    movel([0.342925, -1.240601, -2.657500, -0.814287, 1.570796, 1.913721],accel_mss,speed_ms,0,blend_radius_m)
    movel([0.344869, -1.239133, -2.658265, -0.814990, 1.570796, 1.915665],accel_mss,speed_ms,0,blend_radius_m)
    movel([0.348721, -1.236542, -2.659609, -0.816237, 1.570796, 1.919517],accel_mss,speed_ms,0,blend_radius_m)
    movel([0.352271, -1.234571, -2.660626, -0.817191, 1.570796, 1.923067],accel_mss,speed_ms,0,blend_radius_m)
    movel([0.353507, -1.234027, -2.660906, -0.817455, 1.570796, 1.924303],accel_mss,speed_ms,0,blend_radius_m)
    movel([0.354725, -1.233660, -2.661095, -0.817634, 1.570796, 1.925522],accel_mss,speed_ms,0,blend_radius_m)
    movel([0.355376, -1.233628, -2.661112, -0.817650, 1.570796, 1.926173],accel_mss,speed_ms,0,blend_radius_m)
    movel([0.355877, -1.233849, -2.660998, -0.817542, 1.570796, 1.926673],accel_mss,speed_ms,0,blend_radius_m)
    movel([0.356080, -1.234279, -2.660777, -0.817333, 1.570796, 1.926876],accel_mss,speed_ms,0,blend_radius_m)
    movel([0.355956, -1.234871, -2.660472, -0.817046, 1.570796, 1.926752],accel_mss,speed_ms,0,blend_radius_m)
    movel([0.355650, -1.235547, -2.660124, -0.816719, 1.570796, 1.926446],accel_mss,speed_ms,0,blend_radius_m)
    movel([0.353652, -1.236176, -2.659798, -0.816414, 1.570796, 1.924449],accel_mss,speed_ms,0,blend_radius_m)
    movel([0.351697, -1.236940, -2.659404, -0.816046, 1.570796, 1.922493],accel_mss,speed_ms,0,blend_radius_m)
    movel([0.349633, -1.238027, -2.658840, -0.815522, 1.570796, 1.920429],accel_mss,speed_ms,0,blend_radius_m)
    movel([0.347319, -1.239519, -2.658064, -0.814805, 1.570796, 1.918116],accel_mss,speed_ms,0,blend_radius_m)
    movel([0.344599, -1.241515, -2.657023, -0.813851, 1.570796, 1.915395],accel_mss,speed_ms,0,blend_radius_m)
    movel([0.342464, -1.243303, -2.656086, -0.813000, 1.570796, 1.913260],accel_mss,speed_ms,0,blend_radius_m)
    movel([0.341814, -1.243974, -2.655733, -0.812682, 1.570796, 1.912611],accel_mss,speed_ms,0,blend_radius_m)
    movel([0.341272, -1.244705, -2.655349, -0.812336, 1.570796, 1.912068],accel_mss,speed_ms,0,blend_radius_m)
    movel([0.340309, -1.246556, -2.654371, -0.811462, 1.570796, 1.911105],accel_mss,speed_ms,0,blend_radius_m)
    movel([0.337343, -1.254210, -2.650287, -0.807892, 1.570796, 1.908139],accel_mss,speed_ms,0,blend_radius_m)
    movel([0.336811, -1.255318, -2.649690, -0.807381, 1.570796, 1.907607],accel_mss,speed_ms,0,blend_radius_m)
    movel([0.334705, -1.258850, -2.647777, -0.805762, 1.570796, 1.905501],accel_mss,speed_ms,0,blend_radius_m)
    movel([0.333378, -1.260708, -2.646764, -0.804917, 1.570796, 1.904174],accel_mss,speed_ms,0,blend_radius_m)
    movel([0.331727, -1.262673, -2.645689, -0.804027, 1.570796, 1.902523],accel_mss,speed_ms,0,blend_radius_m)
    movel([0.329183, -1.265435, -2.644170, -0.802785, 1.570796, 1.899980],accel_mss,speed_ms,0,blend_radius_m)
    movel([0.328186, -1.266665, -2.643490, -0.802234, 1.570796, 1.898982],accel_mss,speed_ms,0,blend_radius_m)
    movel([0.327796, -1.267344, -2.643114, -0.801931, 1.570796, 1.898592],accel_mss,speed_ms,0,blend_radius_m)
    movel([0.324763, -1.273372, -2.639750, -0.799266, 1.570796, 1.895559],accel_mss,speed_ms,0,blend_radius_m)
    movel([0.324383, -1.274130, -2.639324, -0.798934, 1.570796, 1.895179],accel_mss,speed_ms,0,blend_radius_m)
    movel([0.324022, -1.275035, -2.638815, -0.798539, 1.570796, 1.894818],accel_mss,speed_ms,0,blend_radius_m)
    movel([0.323870, -1.275151, -2.638750, -0.798489, 1.570796, 1.894666],accel_mss,speed_ms,0,blend_radius_m)
    movel([0.320813, -1.276074, -2.638228, -0.798087, 1.570796, 1.891609],accel_mss,speed_ms,0,blend_radius_m)
    movel([0.319322, -1.276354, -2.638070, -0.797965, 1.570796, 1.890119],accel_mss,speed_ms,0,blend_radius_m)
    movel([0.317735, -1.276515, -2.637979, -0.797895, 1.570796, 1.888532],accel_mss,speed_ms,0,blend_radius_m)
    movel([0.316753, -1.276438, -2.638023, -0.797928, 1.570796, 1.887549],accel_mss,speed_ms,0,blend_radius_m)
    movel([0.316033, -1.276098, -2.638215, -0.798076, 1.570796, 1.886829],accel_mss,speed_ms,0,blend_radius_m)
    movel([0.315335, -1.275398, -2.638610, -0.798381, 1.570796, 1.886132],accel_mss,speed_ms,0,blend_radius_m)
    movel([0.314818, -1.274603, -2.639058, -0.798728, 1.570796, 1.885614],accel_mss,speed_ms,0,blend_radius_m)
    movel([0.314451, -1.273698, -2.639567, -0.799124, 1.570796, 1.885248],accel_mss,speed_ms,0,blend_radius_m)
    movel([0.314212, -1.272638, -2.640162, -0.799588, 1.570796, 1.885009],accel_mss,speed_ms,0,blend_radius_m)
    movel([0.314114, -1.271502, -2.640799, -0.800088, 1.570796, 1.884911],accel_mss,speed_ms,0,blend_radius_m)
    movel([0.314331, -1.268769, -2.642323, -0.801297, 1.570796, 1.885128],accel_mss,speed_ms,0,blend_radius_m)
    movel([0.315111, -1.265451, -2.644161, -0.802778, 1.570796, 1.885907],accel_mss,speed_ms,0,blend_radius_m)
    movel([0.315866, -1.263112, -2.645448, -0.803829, 1.570796, 1.886662],accel_mss,speed_ms,0,blend_radius_m)
    movel([0.316606, -1.261364, -2.646406, -0.804619, 1.570796, 1.887402],accel_mss,speed_ms,0,blend_radius_m)
    movel([0.317785, -1.259161, -2.647608, -0.805620, 1.570796, 1.888582],accel_mss,speed_ms,0,blend_radius_m)
    movel([0.320612, -1.254305, -2.650236, -0.807848, 1.570796, 1.891408],accel_mss,speed_ms,0,blend_radius_m)
    movel([0.326605, -1.243916, -2.655764, -0.812709, 1.570796, 1.897401],accel_mss,speed_ms,0,blend_radius_m)
    movel([0.327796, -1.241515, -2.657023, -0.813851, 1.570796, 1.898593],accel_mss,speed_ms,0,blend_radius_m)
    movel([0.328653, -1.239347, -2.658154, -0.814888, 1.570796, 1.899449],accel_mss,speed_ms,0,blend_radius_m)
    movel([0.329234, -1.237182, -2.659278, -0.815929, 1.570796, 1.900030],accel_mss,speed_ms,0,blend_radius_m)
    movel([0.329337, -1.235501, -2.660147, -0.816741, 1.570796, 1.900134],accel_mss,speed_ms,0,blend_radius_m)
    movel([0.328959, -1.233999, -2.660921, -0.817469, 1.570796, 1.899755],accel_mss,speed_ms,0,blend_radius_m)
    movel([0.327249, -1.231057, -2.662428, -0.818903, 1.570796, 1.898045],accel_mss,speed_ms,0,blend_radius_m)
    movel([0.327023, -1.230500, -2.662713, -0.819176, 1.570796, 1.897820],accel_mss,speed_ms,0,blend_radius_m)
    movel([0.327053, -1.229355, -2.663296, -0.819738, 1.570796, 1.897849],accel_mss,speed_ms,0,blend_radius_m)
    movel([0.327307, -1.228564, -2.663698, -0.820126, 1.570796, 1.898103],accel_mss,speed_ms,0,blend_radius_m)
    movel([0.328348, -1.226520, -2.664734, -0.821135, 1.570796, 1.899144],accel_mss,speed_ms,0,blend_radius_m)
    movel([0.330098, -1.223921, -2.666045, -0.822424, 1.570796, 1.900894],accel_mss,speed_ms,0,blend_radius_m)
    movel([0.332667, -1.220640, -2.667687, -0.824062, 1.570796, 1.903464],accel_mss,speed_ms,0,blend_radius_m)
    movel([0.335094, -1.217632, -2.669182, -0.825575, 1.570796, 1.905891],accel_mss,speed_ms,0,blend_radius_m)
    movel([0.338739, -1.212850, -2.671539, -0.828001, 1.570796, 1.909536],accel_mss,speed_ms,0,blend_radius_m)
    movel([0.338922, -1.212365, -2.671776, -0.828248, 1.570796, 1.909718],accel_mss,speed_ms,0,blend_radius_m)
    movel([0.338575, -1.212129, -2.671891, -0.828368, 1.570796, 1.909372],accel_mss,speed_ms,0,blend_radius_m)
    movel([0.338364, -1.212140, -2.671886, -0.828363, 1.570796, 1.909160],accel_mss,speed_ms,0,blend_radius_m)
    movel([0.337571, -1.212519, -2.671701, -0.828169, 1.570796, 1.908368],accel_mss,speed_ms,0,blend_radius_m)
    movel([0.335837, -1.213970, -2.670989, -0.827430, 1.570796, 1.906634],accel_mss,speed_ms,0,blend_radius_m)
    movel([0.334072, -1.215612, -2.670181, -0.826596, 1.570796, 1.904868],accel_mss,speed_ms,0,blend_radius_m)
    movel([0.332776, -1.217039, -2.669476, -0.825874, 1.570796, 1.903572],accel_mss,speed_ms,0,blend_radius_m)
    movel([0.331388, -1.218851, -2.668578, -0.824960, 1.570796, 1.902184],accel_mss,speed_ms,0,blend_radius_m)
    movel([0.328906, -1.222329, -2.666843, -0.823217, 1.570796, 1.899703],accel_mss,speed_ms,0,blend_radius_m)
    movel([0.325279, -1.227661, -2.664156, -0.820571, 1.570796, 1.896075],accel_mss,speed_ms,0,blend_radius_m)
    movel([0.324263, -1.229633, -2.663155, -0.819601, 1.570796, 1.895059],accel_mss,speed_ms,0,blend_radius_m)
    movel([0.323797, -1.231289, -2.662310, -0.818790, 1.570796, 1.894593],accel_mss,speed_ms,0,blend_radius_m)
    movel([0.323833, -1.232893, -2.661489, -0.818007, 1.570796, 1.894629],accel_mss,speed_ms,0,blend_radius_m)
    movel([0.324369, -1.234718, -2.660551, -0.817120, 1.570796, 1.895165],accel_mss,speed_ms,0,blend_radius_m)
    movel([0.324847, -1.236239, -2.659766, -0.816384, 1.570796, 1.895643],accel_mss,speed_ms,0,blend_radius_m)
    movel([0.325003, -1.237579, -2.659073, -0.815738, 1.570796, 1.895799],accel_mss,speed_ms,0,blend_radius_m)
    movel([0.324852, -1.238985, -2.658342, -0.815062, 1.570796, 1.895648],accel_mss,speed_ms,0,blend_radius_m)
    movel([0.324386, -1.240693, -2.657452, -0.814244, 1.570796, 1.895183],accel_mss,speed_ms,0,blend_radius_m)
    movel([0.322806, -1.244813, -2.655291, -0.812284, 1.570796, 1.893602],accel_mss,speed_ms,0,blend_radius_m)
    movel([0.320559, -1.249674, -2.652716, -0.809999, 1.570796, 1.891355],accel_mss,speed_ms,0,blend_radius_m)
    movel([0.317904, -1.254769, -2.649986, -0.807634, 1.570796, 1.888700],accel_mss,speed_ms,0,blend_radius_m)
    movel([0.313546, -1.262291, -2.645898, -0.804199, 1.570796, 1.884343],accel_mss,speed_ms,0,blend_radius_m)
    movel([0.312665, -1.264271, -2.644811, -0.803307, 1.570796, 1.883462],accel_mss,speed_ms,0,blend_radius_m)
    movel([0.312161, -1.266203, -2.643745, -0.802441, 1.570796, 1.882958],accel_mss,speed_ms,0,blend_radius_m)
    movel([0.311861, -1.268682, -2.642371, -0.801336, 1.570796, 1.882658],accel_mss,speed_ms,0,blend_radius_m)
    movel([0.311715, -1.271688, -2.640695, -0.800006, 1.570796, 1.882512],accel_mss,speed_ms,0,blend_radius_m)
    movel([0.311845, -1.273631, -2.639605, -0.799153, 1.570796, 1.882642],accel_mss,speed_ms,0,blend_radius_m)
    movel([0.312275, -1.275014, -2.638826, -0.798548, 1.570796, 1.883071],accel_mss,speed_ms,0,blend_radius_m)
    movel([0.313063, -1.276155, -2.638183, -0.798051, 1.570796, 1.883860],accel_mss,speed_ms,0,blend_radius_m)
    movel([0.313700, -1.276690, -2.637880, -0.797819, 1.570796, 1.884496],accel_mss,speed_ms,0,blend_radius_m)
    movel([0.314469, -1.277118, -2.637638, -0.797633, 1.570796, 1.885265],accel_mss,speed_ms,0,blend_radius_m)
    movel([0.316829, -1.277817, -2.637241, -0.797330, 1.570796, 1.887625],accel_mss,speed_ms,0,blend_radius_m)
    movel([0.318196, -1.277977, -2.637151, -0.797261, 1.570796, 1.888993],accel_mss,speed_ms,0,blend_radius_m)
    movel([0.319769, -1.277907, -2.637190, -0.797291, 1.570796, 1.890565],accel_mss,speed_ms,0,blend_radius_m)
    movel([0.321417, -1.277620, -2.637353, -0.797415, 1.570796, 1.892213],accel_mss,speed_ms,0,blend_radius_m)
    movel([0.323020, -1.277130, -2.637631, -0.797628, 1.570796, 1.893817],accel_mss,speed_ms,0,blend_radius_m)
    movel([0.324631, -1.276538, -2.637966, -0.797885, 1.570796, 1.895428],accel_mss,speed_ms,0,blend_radius_m)
    movel([0.325024, -1.276490, -2.637993, -0.797906, 1.570796, 1.895820],accel_mss,speed_ms,0,blend_radius_m)
    movel([0.325205, -1.276670, -2.637892, -0.797828, 1.570796, 1.896001],accel_mss,speed_ms,0,blend_radius_m)
    movel([0.325256, -1.277465, -2.637442, -0.797483, 1.570796, 1.896052],accel_mss,speed_ms,0,blend_radius_m)
    movel([0.325263, -1.278170, -2.637041, -0.797178, 1.570796, 1.896059],accel_mss,speed_ms,0,blend_radius_m)
    movel([0.325097, -1.278682, -2.636751, -0.796957, 1.570796, 1.895893],accel_mss,speed_ms,0,blend_radius_m)
    movel([0.324858, -1.278895, -2.636630, -0.796865, 1.570796, 1.895654],accel_mss,speed_ms,0,blend_radius_m)
    movel([0.323615, -1.279507, -2.636281, -0.796601, 1.570796, 1.894411],accel_mss,speed_ms,0,blend_radius_m)
    movel([0.322799, -1.279816, -2.636106, -0.796468, 1.570796, 1.893596],accel_mss,speed_ms,0,blend_radius_m)
    movel([0.322396, -1.281444, -2.635176, -0.795769, 1.570796, 1.893192],accel_mss,speed_ms,0,blend_radius_m)
    movel([0.321882, -1.283464, -2.634019, -0.794906, 1.570796, 1.892679],accel_mss,speed_ms,0,blend_radius_m)
    movel([0.321665, -1.283948, -2.633741, -0.794700, 1.570796, 1.892462],accel_mss,speed_ms,0,blend_radius_m)
    movel([0.321328, -1.284205, -2.633593, -0.794591, 1.570796, 1.892124],accel_mss,speed_ms,0,blend_radius_m)
    movel([0.320496, -1.284406, -2.633477, -0.794506, 1.570796, 1.891293],accel_mss,speed_ms,0,blend_radius_m)
    movel([0.319352, -1.284617, -2.633356, -0.794416, 1.570796, 1.890149],accel_mss,speed_ms,0,blend_radius_m)
    movel([0.319034, -1.286067, -2.632519, -0.793802, 1.570796, 1.889831],accel_mss,speed_ms,0,blend_radius_m)
    movel([0.318968, -1.286670, -2.632171, -0.793548, 1.570796, 1.889764],accel_mss,speed_ms,0,blend_radius_m)
    movel([0.318918, -1.289142, -2.630737, -0.792510, 1.570796, 1.889714],accel_mss,speed_ms,0,blend_radius_m)
    movel([0.317168, -1.289744, -2.630387, -0.792258, 1.570796, 1.887964],accel_mss,speed_ms,0,blend_radius_m)
    movel([0.316818, -1.289909, -2.630291, -0.792189, 1.570796, 1.887614],accel_mss,speed_ms,0,blend_radius_m)
    movel([0.316442, -1.290304, -2.630061, -0.792024, 1.570796, 1.887238],accel_mss,speed_ms,0,blend_radius_m)
    movel([0.316388, -1.290467, -2.629966, -0.791956, 1.570796, 1.887184],accel_mss,speed_ms,0,blend_radius_m)
    movel([0.316505, -1.290778, -2.629785, -0.791827, 1.570796, 1.887301],accel_mss,speed_ms,0,blend_radius_m)
    movel([0.317002, -1.290765, -2.629792, -0.791832, 1.570796, 1.887798],accel_mss,speed_ms,0,blend_radius_m)
    movel([0.319686, -1.289953, -2.630265, -0.792171, 1.570796, 1.890482],accel_mss,speed_ms,0,blend_radius_m)
    movel([0.320071, -1.289692, -2.630418, -0.792280, 1.570796, 1.890868],accel_mss,speed_ms,0,blend_radius_m)
    movel([0.320223, -1.289323, -2.630632, -0.792434, 1.570796, 1.891019],accel_mss,speed_ms,0,blend_radius_m)
    movel([0.320249, -1.289064, -2.630782, -0.792542, 1.570796, 1.891046],accel_mss,speed_ms,0,blend_radius_m)
    movel([0.320099, -1.286560, -2.632235, -0.793594, 1.570796, 1.890895],accel_mss,speed_ms,0,blend_radius_m)
    movel([0.320118, -1.286092, -2.632505, -0.793792, 1.570796, 1.890915],accel_mss,speed_ms,0,blend_radius_m)
    movel([0.320281, -1.285655, -2.632757, -0.793977, 1.570796, 1.891077],accel_mss,speed_ms,0,blend_radius_m)
    movel([0.320489, -1.285544, -2.632822, -0.794024, 1.570796, 1.891285],accel_mss,speed_ms,0,blend_radius_m)
    movel([0.321725, -1.285126, -2.633063, -0.794201, 1.570796, 1.892522],accel_mss,speed_ms,0,blend_radius_m)
    movel([0.322077, -1.284938, -2.633171, -0.794280, 1.570796, 1.892874],accel_mss,speed_ms,0,blend_radius_m)
    movel([0.322644, -1.284448, -2.633453, -0.794488, 1.570796, 1.893440],accel_mss,speed_ms,0,blend_radius_m)
    movel([0.322831, -1.284146, -2.633627, -0.794616, 1.570796, 1.893627],accel_mss,speed_ms,0,blend_radius_m)
    movel([0.323519, -1.281183, -2.635325, -0.795880, 1.570796, 1.894315],accel_mss,speed_ms,0,blend_radius_m)
    movel([0.323687, -1.280709, -2.635596, -0.796084, 1.570796, 1.894484],accel_mss,speed_ms,0,blend_radius_m)
    movel([0.323943, -1.280423, -2.635759, -0.796206, 1.570796, 1.894740],accel_mss,speed_ms,0,blend_radius_m)
    movel([0.324430, -1.280152, -2.635914, -0.796323, 1.570796, 1.895227],accel_mss,speed_ms,0,blend_radius_m)
    movel([0.325816, -1.279294, -2.636403, -0.796693, 1.570796, 1.896612],accel_mss,speed_ms,0,blend_radius_m)
    movel([0.326505, -1.278741, -2.636717, -0.796931, 1.570796, 1.897301],accel_mss,speed_ms,0,blend_radius_m)
    movel([0.326437, -1.275734, -2.638420, -0.798234, 1.570796, 1.897233],accel_mss,speed_ms,0,blend_radius_m)
    movel([0.327765, -1.274947, -2.638865, -0.798578, 1.570796, 1.898561],accel_mss,speed_ms,0,blend_radius_m)
    movel([0.328461, -1.274549, -2.639089, -0.798751, 1.570796, 1.899257],accel_mss,speed_ms,0,blend_radius_m)
    movel([0.335186, -1.270304, -2.641468, -0.800617, 1.570796, 1.905982],accel_mss,speed_ms,0,blend_radius_m)
    movel([0.334839, -1.272294, -2.640355, -0.799740, 1.570796, 1.905635],accel_mss,speed_ms,0,blend_radius_m)
    movel([0.332590, -1.273380, -2.639746, -0.799263, 1.570796, 1.903387],accel_mss,speed_ms,0,blend_radius_m)
    movel([0.330282, -1.274619, -2.639049, -0.798721, 1.570796, 1.901079],accel_mss,speed_ms,0,blend_radius_m)
    movel([0.330077, -1.274797, -2.638949, -0.798643, 1.570796, 1.900873],accel_mss,speed_ms,0,blend_radius_m)
    movel([0.329178, -1.276573, -2.637946, -0.797870, 1.570796, 1.899974],accel_mss,speed_ms,0,blend_radius_m)
    movel([0.328530, -1.277951, -2.637165, -0.797272, 1.570796, 1.899326],accel_mss,speed_ms,0,blend_radius_m)
    movel([0.328008, -1.278732, -2.636722, -0.796935, 1.570796, 1.898804],accel_mss,speed_ms,0,blend_radius_m)
    movel([0.327346, -1.279338, -2.636377, -0.796673, 1.570796, 1.898142],accel_mss,speed_ms,0,blend_radius_m)
    movel([0.326248, -1.280043, -2.635976, -0.796370, 1.570796, 1.897044],accel_mss,speed_ms,0,blend_radius_m)
    movel([0.324771, -1.280902, -2.635486, -0.796001, 1.570796, 1.895567],accel_mss,speed_ms,0,blend_radius_m)
    movel([0.323793, -1.283902, -2.633767, -0.794720, 1.570796, 1.894589],accel_mss,speed_ms,0,blend_radius_m)
    movel([0.323562, -1.284445, -2.633455, -0.794489, 1.570796, 1.894359],accel_mss,speed_ms,0,blend_radius_m)
    movel([0.322925, -1.285601, -2.632788, -0.793999, 1.570796, 1.893721],accel_mss,speed_ms,0,blend_radius_m)
    movel([0.322536, -1.286003, -2.632556, -0.793830, 1.570796, 1.893333],accel_mss,speed_ms,0,blend_radius_m)
    movel([0.320605, -1.287668, -2.631593, -0.793128, 1.570796, 1.891402],accel_mss,speed_ms,0,blend_radius_m)
    movel([0.320516, -1.287805, -2.631514, -0.793070, 1.570796, 1.891312],accel_mss,speed_ms,0,blend_radius_m)
    movel([0.320529, -1.288423, -2.631155, -0.792811, 1.570796, 1.891325],accel_mss,speed_ms,0,blend_radius_m)
    movel([0.320576, -1.288693, -2.630998, -0.792698, 1.570796, 1.891372],accel_mss,speed_ms,0,blend_radius_m)
    movel([0.320625, -1.291004, -2.629653, -0.791733, 1.570796, 1.891421],accel_mss,speed_ms,0,blend_radius_m)
    movel([0.320771, -1.291367, -2.629441, -0.791582, 1.570796, 1.891568],accel_mss,speed_ms,0,blend_radius_m)
    movel([0.321046, -1.291426, -2.629406, -0.791557, 1.570796, 1.891842],accel_mss,speed_ms,0,blend_radius_m)
    movel([0.321425, -1.291226, -2.629523, -0.791640, 1.570796, 1.892222],accel_mss,speed_ms,0,blend_radius_m)
    movel([0.322031, -1.290877, -2.629727, -0.791785, 1.570796, 1.892827],accel_mss,speed_ms,0,blend_radius_m)
    movel([0.317945, -1.294449, -2.627633, -0.790307, 1.570796, 1.888741],accel_mss,speed_ms,0,blend_radius_m)
    movel([0.314705, -1.297568, -2.625792, -0.789029, 1.570796, 1.885501],accel_mss,speed_ms,0,blend_radius_m)
    movel([0.311613, -1.300747, -2.623903, -0.787739, 1.570796, 1.882409],accel_mss,speed_ms,0,blend_radius_m)
    movel([0.309536, -1.303153, -2.622464, -0.786772, 1.570796, 1.880332],accel_mss,speed_ms,0,blend_radius_m)
    movel([0.307881, -1.305516, -2.621043, -0.785829, 1.570796, 1.878677],accel_mss,speed_ms,0,blend_radius_m)
    movel([0.307303, -1.306574, -2.620406, -0.785410, 1.570796, 1.878099],accel_mss,speed_ms,0,blend_radius_m)
    movel([0.306855, -1.307631, -2.619766, -0.784992, 1.570796, 1.877651],accel_mss,speed_ms,0,blend_radius_m)
    movel([0.306618, -1.308486, -2.619248, -0.784655, 1.570796, 1.877415],accel_mss,speed_ms,0,blend_radius_m)
    movel([0.306533, -1.309299, -2.618754, -0.784335, 1.570796, 1.877329],accel_mss,speed_ms,0,blend_radius_m)
    movel([0.306634, -1.309898, -2.618390, -0.784100, 1.570796, 1.877431],accel_mss,speed_ms,0,blend_radius_m)
    movel([0.306944, -1.310362, -2.618108, -0.783919, 1.570796, 1.877741],accel_mss,speed_ms,0,blend_radius_m)
    movel([0.307420, -1.310668, -2.617922, -0.783799, 1.570796, 1.878216],accel_mss,speed_ms,0,blend_radius_m)
    movel([0.307844, -1.310614, -2.617955, -0.783820, 1.570796, 1.878640],accel_mss,speed_ms,0,blend_radius_m)
    movel([0.308283, -1.310234, -2.618186, -0.783969, 1.570796, 1.879079],accel_mss,speed_ms,0,blend_radius_m)
    movel([0.309618, -1.308138, -2.619459, -0.784792, 1.570796, 1.880414],accel_mss,speed_ms,0,blend_radius_m)
    movel([0.309710, -1.308359, -2.619325, -0.784705, 1.570796, 1.880506],accel_mss,speed_ms,0,blend_radius_m)
    movel([0.309632, -1.308862, -2.619020, -0.784507, 1.570796, 1.880428],accel_mss,speed_ms,0,blend_radius_m)
    movel([0.309835, -1.310236, -2.618185, -0.783968, 1.570796, 1.880632],accel_mss,speed_ms,0,blend_radius_m)
    movel([0.310053, -1.310680, -2.617915, -0.783795, 1.570796, 1.880849],accel_mss,speed_ms,0,blend_radius_m)
    movel([0.310331, -1.310909, -2.617775, -0.783705, 1.570796, 1.881127],accel_mss,speed_ms,0,blend_radius_m)
    movel([0.310697, -1.310970, -2.617737, -0.783681, 1.570796, 1.881493],accel_mss,speed_ms,0,blend_radius_m)
    movel([0.311102, -1.310852, -2.617810, -0.783727, 1.570796, 1.881898],accel_mss,speed_ms,0,blend_radius_m)
    movel([0.311497, -1.310578, -2.617977, -0.783834, 1.570796, 1.882293],accel_mss,speed_ms,0,blend_radius_m)
    movel([0.313004, -1.308779, -2.619070, -0.784539, 1.570796, 1.883800],accel_mss,speed_ms,0,blend_radius_m)
    movel([0.314562, -1.306982, -2.620159, -0.785248, 1.570796, 1.885358],accel_mss,speed_ms,0,blend_radius_m)
    movel([0.316271, -1.305388, -2.621121, -0.785880, 1.570796, 1.887067],accel_mss,speed_ms,0,blend_radius_m)
    movel([0.318253, -1.303895, -2.622019, -0.786475, 1.570796, 1.889049],accel_mss,speed_ms,0,blend_radius_m)
    movel([0.320643, -1.302395, -2.622918, -0.787076, 1.570796, 1.891440],accel_mss,speed_ms,0,blend_radius_m)
    movel([0.322090, -1.301513, -2.623446, -0.787431, 1.570796, 1.892887],accel_mss,speed_ms,0,blend_radius_m)
    movel([0.323181, -1.300731, -2.623912, -0.787746, 1.570796, 1.893977],accel_mss,speed_ms,0,blend_radius_m)
    movel([0.324024, -1.299978, -2.624361, -0.788050, 1.570796, 1.894820],accel_mss,speed_ms,0,blend_radius_m)
    movel([0.324700, -1.299185, -2.624833, -0.788371, 1.570796, 1.895496],accel_mss,speed_ms,0,blend_radius_m)
    movel([0.325241, -1.298267, -2.625378, -0.788744, 1.570796, 1.896038],accel_mss,speed_ms,0,blend_radius_m)
    movel([0.326301, -1.295864, -2.626800, -0.789725, 1.570796, 1.897097],accel_mss,speed_ms,0,blend_radius_m)
    movel([0.327337, -1.293401, -2.628249, -0.790739, 1.570796, 1.898134],accel_mss,speed_ms,0,blend_radius_m)
    movel([0.327468, -1.292744, -2.628635, -0.791011, 1.570796, 1.898264],accel_mss,speed_ms,0,blend_radius_m)
    movel([0.327010, -1.292596, -2.628721, -0.791072, 1.570796, 1.897806],accel_mss,speed_ms,0,blend_radius_m)
    movel([0.326728, -1.292738, -2.628638, -0.791013, 1.570796, 1.897524],accel_mss,speed_ms,0,blend_radius_m)
    movel([0.326507, -1.292983, -2.628494, -0.790911, 1.570796, 1.897303],accel_mss,speed_ms,0,blend_radius_m)
    movel([0.326260, -1.293466, -2.628211, -0.790712, 1.570796, 1.897057],accel_mss,speed_ms,0,blend_radius_m)
    movel([0.324268, -1.298014, -2.625528, -0.788847, 1.570796, 1.895064],accel_mss,speed_ms,0,blend_radius_m)
    movel([0.323726, -1.298957, -2.624968, -0.788464, 1.570796, 1.894522],accel_mss,speed_ms,0,blend_radius_m)
    movel([0.323219, -1.299594, -2.624590, -0.788205, 1.570796, 1.894016],accel_mss,speed_ms,0,blend_radius_m)
    movel([0.322852, -1.299911, -2.624401, -0.788077, 1.570796, 1.893648],accel_mss,speed_ms,0,blend_radius_m)
    movel([0.320257, -1.301603, -2.623392, -0.787394, 1.570796, 1.891053],accel_mss,speed_ms,0,blend_radius_m)
    movel([0.317454, -1.303416, -2.622306, -0.786667, 1.570796, 1.888250],accel_mss,speed_ms,0,blend_radius_m)
    movel([0.315089, -1.305277, -2.621188, -0.785924, 1.570796, 1.885885],accel_mss,speed_ms,0,blend_radius_m)
    movel([0.313132, -1.307206, -2.620023, -0.785159, 1.570796, 1.883929],accel_mss,speed_ms,0,blend_radius_m)
    movel([0.311547, -1.309229, -2.618797, -0.784363, 1.570796, 1.882344],accel_mss,speed_ms,0,blend_radius_m)
    movel([0.311164, -1.309800, -2.618450, -0.784139, 1.570796, 1.881960],accel_mss,speed_ms,0,blend_radius_m)
    movel([0.310958, -1.309434, -2.618672, -0.784282, 1.570796, 1.881754],accel_mss,speed_ms,0,blend_radius_m)
    movel([0.310806, -1.308882, -2.619008, -0.784499, 1.570796, 1.881602],accel_mss,speed_ms,0,blend_radius_m)
    movel([0.310862, -1.308093, -2.619487, -0.784810, 1.570796, 1.881658],accel_mss,speed_ms,0,blend_radius_m)
    movel([0.311103, -1.307181, -2.620039, -0.785170, 1.570796, 1.881900],accel_mss,speed_ms,0,blend_radius_m)
    movel([0.311870, -1.305620, -2.620981, -0.785788, 1.570796, 1.882666],accel_mss,speed_ms,0,blend_radius_m)
    movel([0.312202, -1.305169, -2.621253, -0.785967, 1.570796, 1.882998],accel_mss,speed_ms,0,blend_radius_m)
    movel([0.313355, -1.304117, -2.621885, -0.786386, 1.570796, 1.884152],accel_mss,speed_ms,0,blend_radius_m)
    movel([0.314742, -1.303078, -2.622509, -0.786802, 1.570796, 1.885538],accel_mss,speed_ms,0,blend_radius_m)
    movel([0.316222, -1.302150, -2.623065, -0.787174, 1.570796, 1.887019],accel_mss,speed_ms,0,blend_radius_m)
    movel([0.317816, -1.301322, -2.623560, -0.787507, 1.570796, 1.888613],accel_mss,speed_ms,0,blend_radius_m)
    movel([0.321143, -1.299907, -2.624404, -0.788079, 1.570796, 1.891939],accel_mss,speed_ms,0,blend_radius_m)
    movel([0.321780, -1.299609, -2.624581, -0.788199, 1.570796, 1.892576],accel_mss,speed_ms,0,blend_radius_m)
    movel([0.322460, -1.299066, -2.624903, -0.788419, 1.570796, 1.893257],accel_mss,speed_ms,0,blend_radius_m)
    movel([0.322781, -1.298643, -2.625155, -0.788591, 1.570796, 1.893577],accel_mss,speed_ms,0,blend_radius_m)
    movel([0.325964, -1.293186, -2.628375, -0.790828, 1.570796, 1.896760],accel_mss,speed_ms,0,blend_radius_m)
    movel([0.326690, -1.291543, -2.629337, -0.791508, 1.570796, 1.897486],accel_mss,speed_ms,0,blend_radius_m)
    movel([0.326759, -1.291157, -2.629563, -0.791669, 1.570796, 1.897555],accel_mss,speed_ms,0,blend_radius_m)
    movel([0.326656, -1.290909, -2.629708, -0.791772, 1.570796, 1.897453],accel_mss,speed_ms,0,blend_radius_m)
    movel([0.326423, -1.290864, -2.629734, -0.791791, 1.570796, 1.897220],accel_mss,speed_ms,0,blend_radius_m)
    movel([0.326121, -1.291020, -2.629643, -0.791726, 1.570796, 1.896918],accel_mss,speed_ms,0,blend_radius_m)
    movel([0.325974, -1.291191, -2.629543, -0.791655, 1.570796, 1.896770],accel_mss,speed_ms,0,blend_radius_m)
    movel([0.325499, -1.292006, -2.629067, -0.791316, 1.570796, 1.896296],accel_mss,speed_ms,0,blend_radius_m)
    movel([0.322492, -1.297479, -2.625845, -0.789065, 1.570796, 1.893288],accel_mss,speed_ms,0,blend_radius_m)
    movel([0.321971, -1.298129, -2.625460, -0.788800, 1.570796, 1.892767],accel_mss,speed_ms,0,blend_radius_m)
    movel([0.321361, -1.298657, -2.625147, -0.788586, 1.570796, 1.892157],accel_mss,speed_ms,0,blend_radius_m)
    movel([0.320584, -1.299114, -2.624875, -0.788400, 1.570796, 1.891380],accel_mss,speed_ms,0,blend_radius_m)
    movel([0.319549, -1.299559, -2.624610, -0.788219, 1.570796, 1.890346],accel_mss,speed_ms,0,blend_radius_m)
    movel([0.317931, -1.300249, -2.624200, -0.787940, 1.570796, 1.888727],accel_mss,speed_ms,0,blend_radius_m)
    movel([0.316327, -1.301072, -2.623709, -0.787608, 1.570796, 1.887123],accel_mss,speed_ms,0,blend_radius_m)
    movel([0.314798, -1.302007, -2.623150, -0.787232, 1.570796, 1.885594],accel_mss,speed_ms,0,blend_radius_m)
    movel([0.313325, -1.303059, -2.622520, -0.786810, 1.570796, 1.884122],accel_mss,speed_ms,0,blend_radius_m)
    movel([0.311974, -1.304185, -2.621845, -0.786359, 1.570796, 1.882770],accel_mss,speed_ms,0,blend_radius_m)
    movel([0.310714, -1.305403, -2.621112, -0.785874, 1.570796, 1.881511],accel_mss,speed_ms,0,blend_radius_m)
    movel([0.309608, -1.306657, -2.620355, -0.785377, 1.570796, 1.880404],accel_mss,speed_ms,0,blend_radius_m)
    movel([0.307970, -1.308883, -2.619007, -0.784499, 1.570796, 1.878766],accel_mss,speed_ms,0,blend_radius_m)
    movel([0.307710, -1.309189, -2.618821, -0.784378, 1.570796, 1.878506],accel_mss,speed_ms,0,blend_radius_m)
    movel([0.307514, -1.308971, -2.618954, -0.784464, 1.570796, 1.878310],accel_mss,speed_ms,0,blend_radius_m)
    movel([0.307902, -1.307511, -2.619839, -0.785039, 1.570796, 1.878698],accel_mss,speed_ms,0,blend_radius_m)
    movel([0.308286, -1.306650, -2.620360, -0.785380, 1.570796, 1.879083],accel_mss,speed_ms,0,blend_radius_m)
    movel([0.309357, -1.304875, -2.621430, -0.786084, 1.570796, 1.880153],accel_mss,speed_ms,0,blend_radius_m)
    movel([0.310889, -1.302894, -2.622619, -0.786876, 1.570796, 1.881686],accel_mss,speed_ms,0,blend_radius_m)
    movel([0.313080, -1.300464, -2.624072, -0.787854, 1.570796, 1.883877],accel_mss,speed_ms,0,blend_radius_m)
    movel([0.316245, -1.297249, -2.625981, -0.789159, 1.570796, 1.887041],accel_mss,speed_ms,0,blend_radius_m)
    movel([0.318267, -1.295330, -2.627115, -0.789944, 1.570796, 1.889063],accel_mss,speed_ms,0,blend_radius_m)
    movel([0.320323, -1.293542, -2.628166, -0.790681, 1.570796, 1.891120],accel_mss,speed_ms,0,blend_radius_m)
    movel([0.322292, -1.291992, -2.629075, -0.791322, 1.570796, 1.893089],accel_mss,speed_ms,0,blend_radius_m)
    movel([0.324033, -1.290798, -2.629773, -0.791818, 1.570796, 1.894829],accel_mss,speed_ms,0,blend_radius_m)
    movel([0.326419, -1.289247, -2.630676, -0.792465, 1.570796, 1.897215],accel_mss,speed_ms,0,blend_radius_m)
    movel([0.326571, -1.289012, -2.630813, -0.792564, 1.570796, 1.897367],accel_mss,speed_ms,0,blend_radius_m)
    movel([0.326529, -1.288772, -2.630953, -0.792665, 1.570796, 1.897325],accel_mss,speed_ms,0,blend_radius_m)
    movel([0.326265, -1.288629, -2.631035, -0.792724, 1.570796, 1.897061],accel_mss,speed_ms,0,blend_radius_m)
    movel([0.325881, -1.288688, -2.631001, -0.792700, 1.570796, 1.896677],accel_mss,speed_ms,0,blend_radius_m)
    movel([0.325245, -1.289001, -2.630819, -0.792569, 1.570796, 1.896041],accel_mss,speed_ms,0,blend_radius_m)
    movel([0.323486, -1.290082, -2.630190, -0.792117, 1.570796, 1.894283],accel_mss,speed_ms,0,blend_radius_m)
    movel([0.323015, -1.290364, -2.630026, -0.791999, 1.570796, 1.893811],accel_mss,speed_ms,0,blend_radius_m)
    movel([0.322566, -1.290595, -2.629891, -0.791903, 1.570796, 1.893362],accel_mss,speed_ms,0,blend_radius_m)
    movel([0.322581, -1.290460, -2.629970, -0.791959, 1.570796, 1.893377],accel_mss,speed_ms,0,blend_radius_m)
    movel([0.324238, -1.287850, -2.631488, -0.793051, 1.570796, 1.895035],accel_mss,speed_ms,0,blend_radius_m)
    movel([0.325747, -1.285504, -2.632845, -0.794041, 1.570796, 1.896543],accel_mss,speed_ms,0,blend_radius_m)
    movel([0.327501, -1.283042, -2.634261, -0.795086, 1.570796, 1.898298],accel_mss,speed_ms,0,blend_radius_m)
    movel([0.328546, -1.281758, -2.634997, -0.795634, 1.570796, 1.899342],accel_mss,speed_ms,0,blend_radius_m)
    movel([0.330499, -1.279591, -2.636233, -0.796564, 1.570796, 1.901296],accel_mss,speed_ms,0,blend_radius_m)
    movel([0.331023, -1.279101, -2.636512, -0.796776, 1.570796, 1.901819],accel_mss,speed_ms,0,blend_radius_m)
    movel([0.337924, -1.273196, -2.639849, -0.799343, 1.570796, 1.908721],accel_mss,speed_ms,0,blend_radius_m)
    movel([0.339035, -1.272173, -2.640423, -0.799793, 1.570796, 1.909832],accel_mss,speed_ms,0,blend_radius_m)
    movel([0.340660, -1.270300, -2.641470, -0.800619, 1.570796, 1.911456],accel_mss,speed_ms,0,blend_radius_m)
    movel([0.341728, -1.268826, -2.642291, -0.801272, 1.570796, 1.912524],accel_mss,speed_ms,0,blend_radius_m)
    movel([0.343334, -1.266218, -2.643737, -0.802434, 1.570796, 1.914131],accel_mss,speed_ms,0,blend_radius_m)
    movel([0.343530, -1.265850, -2.643940, -0.802599, 1.570796, 1.914327],accel_mss,speed_ms,0,blend_radius_m)
    movel([0.344082, -1.265081, -2.644365, -0.802943, 1.570796, 1.914878],accel_mss,speed_ms,0,blend_radius_m)
    movel([0.344815, -1.264701, -2.644574, -0.803114, 1.570796, 1.915611],accel_mss,speed_ms,0,blend_radius_m)
    movel([0.346399, -1.264254, -2.644820, -0.803315, 1.570796, 1.917195],accel_mss,speed_ms,0,blend_radius_m)
    movel([0.348049, -1.263892, -2.645019, -0.803477, 1.570796, 1.918846],accel_mss,speed_ms,0,blend_radius_m)
    movel([0.349307, -1.263755, -2.645095, -0.803539, 1.570796, 1.920104],accel_mss,speed_ms,0,blend_radius_m)
    movel([0.351720, -1.263668, -2.645142, -0.803578, 1.570796, 1.922516],accel_mss,speed_ms,0,blend_radius_m)
    movel([0.353758, -1.263475, -2.645249, -0.803665, 1.570796, 1.924554],accel_mss,speed_ms,0,blend_radius_m)
    movel([0.354469, -1.263278, -2.645357, -0.803754, 1.570796, 1.925265],accel_mss,speed_ms,0,blend_radius_m)
    movel([0.355370, -1.262854, -2.645590, -0.803945, 1.570796, 1.926167],accel_mss,speed_ms,0,blend_radius_m)
    movel([0.356366, -1.262188, -2.645955, -0.804246, 1.570796, 1.927163],accel_mss,speed_ms,0,blend_radius_m)
    movel([0.357266, -1.261419, -2.646376, -0.804594, 1.570796, 1.928062],accel_mss,speed_ms,0,blend_radius_m)
    movel([0.357880, -1.260692, -2.646773, -0.804924, 1.570796, 1.928676],accel_mss,speed_ms,0,blend_radius_m)
    movel([0.358330, -1.259858, -2.647228, -0.805303, 1.570796, 1.929127],accel_mss,speed_ms,0,blend_radius_m)
    movel([0.358354, -1.259638, -2.647348, -0.805403, 1.570796, 1.929150],accel_mss,speed_ms,0,blend_radius_m)
    movel([0.358229, -1.259509, -2.647418, -0.805462, 1.570796, 1.929026],accel_mss,speed_ms,0,blend_radius_m)
    movel([0.357635, -1.259557, -2.647392, -0.805440, 1.570796, 1.928432],accel_mss,speed_ms,0,blend_radius_m)
    movel([0.356291, -1.260149, -2.647069, -0.805171, 1.570796, 1.927088],accel_mss,speed_ms,0,blend_radius_m)
    movel([0.355411, -1.260533, -2.646860, -0.804996, 1.570796, 1.926207],accel_mss,speed_ms,0,blend_radius_m)
    movel([0.353833, -1.260857, -2.646683, -0.804849, 1.570796, 1.924629],accel_mss,speed_ms,0,blend_radius_m)
    movel([0.351708, -1.261032, -2.646588, -0.804770, 1.570796, 1.922505],accel_mss,speed_ms,0,blend_radius_m)
    movel([0.347995, -1.261470, -2.646348, -0.804571, 1.570796, 1.918792],accel_mss,speed_ms,0,blend_radius_m)
    movel([0.347302, -1.261647, -2.646251, -0.804491, 1.570796, 1.918098],accel_mss,speed_ms,0,blend_radius_m)
    movel([0.346143, -1.261915, -2.646105, -0.804370, 1.570796, 1.916939],accel_mss,speed_ms,0,blend_radius_m)
    movel([0.347217, -1.261402, -2.646385, -0.804602, 1.570796, 1.918014],accel_mss,speed_ms,0,blend_radius_m)
    movel([0.347469, -1.261203, -2.646494, -0.804692, 1.570796, 1.918265],accel_mss,speed_ms,0,blend_radius_m)
    movel([0.348062, -1.260057, -2.647119, -0.805212, 1.570796, 1.918858],accel_mss,speed_ms,0,blend_radius_m)
    movel([0.348945, -1.258428, -2.648006, -0.805955, 1.570796, 1.919741],accel_mss,speed_ms,0,blend_radius_m)
    movel([0.349955, -1.257198, -2.648673, -0.806517, 1.570796, 1.920751],accel_mss,speed_ms,0,blend_radius_m)
    movel([0.351344, -1.256104, -2.649266, -0.807020, 1.570796, 1.922141],accel_mss,speed_ms,0,blend_radius_m)
    movel([0.354660, -1.254202, -2.650291, -0.807895, 1.570796, 1.925456],accel_mss,speed_ms,0,blend_radius_m)
    movel([0.355744, -1.253524, -2.650656, -0.808209, 1.570796, 1.926540],accel_mss,speed_ms,0,blend_radius_m)
    movel([0.358178, -1.251746, -2.651610, -0.809034, 1.570796, 1.928974],accel_mss,speed_ms,0,blend_radius_m)
    movel([0.360077, -1.250337, -2.652363, -0.809690, 1.570796, 1.930873],accel_mss,speed_ms,0,blend_radius_m)
    movel([0.361752, -1.249264, -2.652934, -0.810191, 1.570796, 1.932548],accel_mss,speed_ms,0,blend_radius_m)
    movel([0.363207, -1.248516, -2.653332, -0.810541, 1.570796, 1.934003],accel_mss,speed_ms,0,blend_radius_m)
    movel([0.364430, -1.248103, -2.653552, -0.810735, 1.570796, 1.935227],accel_mss,speed_ms,0,blend_radius_m)
    movel([0.365326, -1.247905, -2.653656, -0.810827, 1.570796, 1.936123],accel_mss,speed_ms,0,blend_radius_m)
    movel([0.364600, -1.248375, -2.653407, -0.810607, 1.570796, 1.935397],accel_mss,speed_ms,0,blend_radius_m)
    movel([0.363917, -1.248860, -2.653149, -0.810380, 1.570796, 1.934713],accel_mss,speed_ms,0,blend_radius_m)
    movel([0.363580, -1.249221, -2.652957, -0.810211, 1.570796, 1.934376],accel_mss,speed_ms,0,blend_radius_m)
    movel([0.363466, -1.249563, -2.652775, -0.810051, 1.570796, 1.934262],accel_mss,speed_ms,0,blend_radius_m)
    movel([0.363555, -1.249959, -2.652564, -0.809866, 1.570796, 1.934352],accel_mss,speed_ms,0,blend_radius_m)
    movel([0.363627, -1.250390, -2.652334, -0.809665, 1.570796, 1.934423],accel_mss,speed_ms,0,blend_radius_m)
    movel([0.363434, -1.250697, -2.652170, -0.809522, 1.570796, 1.934230],accel_mss,speed_ms,0,blend_radius_m)
    movel([0.362929, -1.250944, -2.652038, -0.809406, 1.570796, 1.933725],accel_mss,speed_ms,0,blend_radius_m)
    movel([0.361806, -1.251216, -2.651893, -0.809280, 1.570796, 1.932602],accel_mss,speed_ms,0,blend_radius_m)
    movel([0.361216, -1.251361, -2.651815, -0.809212, 1.570796, 1.932012],accel_mss,speed_ms,0,blend_radius_m)
    movel([0.359689, -1.251903, -2.651525, -0.808960, 1.570796, 1.930485],accel_mss,speed_ms,0,blend_radius_m)
    movel([0.358885, -1.252395, -2.651262, -0.808732, 1.570796, 1.929682],accel_mss,speed_ms,0,blend_radius_m)
    movel([0.357422, -1.253606, -2.650612, -0.808171, 1.570796, 1.928219],accel_mss,speed_ms,0,blend_radius_m)
    movel([0.357149, -1.254014, -2.650393, -0.807982, 1.570796, 1.927946],accel_mss,speed_ms,0,blend_radius_m)
    movel([0.357131, -1.254366, -2.650203, -0.807820, 1.570796, 1.927927],accel_mss,speed_ms,0,blend_radius_m)
    movel([0.357355, -1.254463, -2.650151, -0.807775, 1.570796, 1.928151],accel_mss,speed_ms,0,blend_radius_m)
    movel([0.357869, -1.254246, -2.650268, -0.807876, 1.570796, 1.928666],accel_mss,speed_ms,0,blend_radius_m)
    movel([0.358661, -1.253697, -2.650563, -0.808129, 1.570796, 1.929457],accel_mss,speed_ms,0,blend_radius_m)
    movel([0.360116, -1.252790, -2.651050, -0.808549, 1.570796, 1.930912],accel_mss,speed_ms,0,blend_radius_m)
    movel([0.360865, -1.252538, -2.651185, -0.808666, 1.570796, 1.931661],accel_mss,speed_ms,0,blend_radius_m)
    movel([0.363410, -1.251855, -2.651551, -0.808983, 1.570796, 1.934207],accel_mss,speed_ms,0,blend_radius_m)
    movel([0.363833, -1.251631, -2.651671, -0.809087, 1.570796, 1.934629],accel_mss,speed_ms,0,blend_radius_m)
    movel([0.364528, -1.250957, -2.652032, -0.809401, 1.570796, 1.935324],accel_mss,speed_ms,0,blend_radius_m)
    movel([0.364731, -1.250566, -2.652240, -0.809583, 1.570796, 1.935528],accel_mss,speed_ms,0,blend_radius_m)
    movel([0.364985, -1.249525, -2.652795, -0.810069, 1.570796, 1.935782],accel_mss,speed_ms,0,blend_radius_m)
    movel([0.365181, -1.249233, -2.652951, -0.810205, 1.570796, 1.935977],accel_mss,speed_ms,0,blend_radius_m)
    movel([0.366684, -1.248398, -2.653395, -0.810596, 1.570796, 1.937480],accel_mss,speed_ms,0,blend_radius_m)
    movel([0.367580, -1.248064, -2.653572, -0.810753, 1.570796, 1.938377],accel_mss,speed_ms,0,blend_radius_m)
    movel([0.368267, -1.247940, -2.653638, -0.810811, 1.570796, 1.939063],accel_mss,speed_ms,0,blend_radius_m)
    movel([0.368501, -1.247999, -2.653607, -0.810783, 1.570796, 1.939297],accel_mss,speed_ms,0,blend_radius_m)
    movel([0.370616, -1.249162, -2.652988, -0.810238, 1.570796, 1.941412],accel_mss,speed_ms,0,blend_radius_m)
    movel([0.371633, -1.249698, -2.652703, -0.809988, 1.570796, 1.942429],accel_mss,speed_ms,0,blend_radius_m)
    movel([0.372299, -1.250229, -2.652420, -0.809740, 1.570796, 1.943095],accel_mss,speed_ms,0,blend_radius_m)
    movel([0.372643, -1.250747, -2.652144, -0.809499, 1.570796, 1.943440],accel_mss,speed_ms,0,blend_radius_m)
    movel([0.372623, -1.251242, -2.651879, -0.809268, 1.570796, 1.943419],accel_mss,speed_ms,0,blend_radius_m)
    movel([0.372214, -1.251826, -2.651567, -0.808996, 1.570796, 1.943011],accel_mss,speed_ms,0,blend_radius_m)
    movel([0.370206, -1.253650, -2.650588, -0.808151, 1.570796, 1.941003],accel_mss,speed_ms,0,blend_radius_m)
    movel([0.368211, -1.255383, -2.649655, -0.807351, 1.570796, 1.939007],accel_mss,speed_ms,0,blend_radius_m)
    movel([0.366962, -1.256306, -2.649156, -0.806926, 1.570796, 1.937758],accel_mss,speed_ms,0,blend_radius_m)
    movel([0.365877, -1.256870, -2.648851, -0.806668, 1.570796, 1.936673],accel_mss,speed_ms,0,blend_radius_m)
    movel([0.364763, -1.257194, -2.648676, -0.806519, 1.570796, 1.935559],accel_mss,speed_ms,0,blend_radius_m)
    movel([0.363726, -1.257250, -2.648646, -0.806494, 1.570796, 1.934522],accel_mss,speed_ms,0,blend_radius_m)
    movel([0.362348, -1.256846, -2.648864, -0.806679, 1.570796, 1.933144],accel_mss,speed_ms,0,blend_radius_m)
    movel([0.361912, -1.256830, -2.648873, -0.806686, 1.570796, 1.932709],accel_mss,speed_ms,0,blend_radius_m)
    movel([0.361591, -1.256977, -2.648793, -0.806619, 1.570796, 1.932387],accel_mss,speed_ms,0,blend_radius_m)
    movel([0.361381, -1.257253, -2.648644, -0.806492, 1.570796, 1.932178],accel_mss,speed_ms,0,blend_radius_m)
    movel([0.361336, -1.257546, -2.648485, -0.806358, 1.570796, 1.932132],accel_mss,speed_ms,0,blend_radius_m)
    movel([0.361428, -1.257767, -2.648365, -0.806257, 1.570796, 1.932225],accel_mss,speed_ms,0,blend_radius_m)
    movel([0.362026, -1.258183, -2.648139, -0.806067, 1.570796, 1.932822],accel_mss,speed_ms,0,blend_radius_m)
    movel([0.362965, -1.258423, -2.648009, -0.805957, 1.570796, 1.933761],accel_mss,speed_ms,0,blend_radius_m)
    movel([0.364065, -1.258419, -2.648011, -0.805959, 1.570796, 1.934861],accel_mss,speed_ms,0,blend_radius_m)
    movel([0.365032, -1.258233, -2.648112, -0.806044, 1.570796, 1.935828],accel_mss,speed_ms,0,blend_radius_m)
    movel([0.365993, -1.257889, -2.648299, -0.806201, 1.570796, 1.936790],accel_mss,speed_ms,0,blend_radius_m)
    movel([0.366972, -1.257376, -2.648577, -0.806436, 1.570796, 1.937768],accel_mss,speed_ms,0,blend_radius_m)
    movel([0.367999, -1.256681, -2.648954, -0.806755, 1.570796, 1.938795],accel_mss,speed_ms,0,blend_radius_m)
    movel([0.368656, -1.256206, -2.649210, -0.806972, 1.570796, 1.939453],accel_mss,speed_ms,0,blend_radius_m)
    movel([0.368859, -1.256161, -2.649235, -0.806993, 1.570796, 1.939655],accel_mss,speed_ms,0,blend_radius_m)
    movel([0.368934, -1.256308, -2.649155, -0.806925, 1.570796, 1.939730],accel_mss,speed_ms,0,blend_radius_m)
    movel([0.368831, -1.257017, -2.648772, -0.806601, 1.570796, 1.939627],accel_mss,speed_ms,0,blend_radius_m)
    movel([0.368626, -1.257710, -2.648396, -0.806283, 1.570796, 1.939422],accel_mss,speed_ms,0,blend_radius_m)
    movel([0.368272, -1.258253, -2.648101, -0.806035, 1.570796, 1.939068],accel_mss,speed_ms,0,blend_radius_m)
    movel([0.367693, -1.258745, -2.647834, -0.805810, 1.570796, 1.938489],accel_mss,speed_ms,0,blend_radius_m)
    movel([0.366237, -1.259567, -2.647387, -0.805436, 1.570796, 1.937033],accel_mss,speed_ms,0,blend_radius_m)
    movel([0.365755, -1.259843, -2.647236, -0.805310, 1.570796, 1.936551],accel_mss,speed_ms,0,blend_radius_m)
    movel([0.364730, -1.260577, -2.646836, -0.804976, 1.570796, 1.935526],accel_mss,speed_ms,0,blend_radius_m)
    movel([0.364325, -1.260845, -2.646689, -0.804854, 1.570796, 1.935121],accel_mss,speed_ms,0,blend_radius_m)
    movel([0.362762, -1.261684, -2.646231, -0.804474, 1.570796, 1.933558],accel_mss,speed_ms,0,blend_radius_m)
    movel([0.362247, -1.261816, -2.646159, -0.804414, 1.570796, 1.933044],accel_mss,speed_ms,0,blend_radius_m)
    movel([0.361005, -1.261953, -2.646084, -0.804353, 1.570796, 1.931802],accel_mss,speed_ms,0,blend_radius_m)
    movel([0.360394, -1.261953, -2.646084, -0.804353, 1.570796, 1.931190],accel_mss,speed_ms,0,blend_radius_m)
    movel([0.358488, -1.261740, -2.646200, -0.804449, 1.570796, 1.929284],accel_mss,speed_ms,0,blend_radius_m)
    movel([0.358253, -1.261818, -2.646157, -0.804413, 1.570796, 1.929050],accel_mss,speed_ms,0,blend_radius_m)
    movel([0.357741, -1.262213, -2.645941, -0.804235, 1.570796, 1.928537],accel_mss,speed_ms,0,blend_radius_m)
    movel([0.357740, -1.262625, -2.645715, -0.804049, 1.570796, 1.928536],accel_mss,speed_ms,0,blend_radius_m)
    movel([0.358143, -1.262900, -2.645565, -0.803925, 1.570796, 1.928939],accel_mss,speed_ms,0,blend_radius_m)
    movel([0.359018, -1.263072, -2.645470, -0.803847, 1.570796, 1.929814],accel_mss,speed_ms,0,blend_radius_m)
    movel([0.360121, -1.263136, -2.645435, -0.803818, 1.570796, 1.930918],accel_mss,speed_ms,0,blend_radius_m)
    movel([0.362353, -1.263005, -2.645507, -0.803877, 1.570796, 1.933149],accel_mss,speed_ms,0,blend_radius_m)
    movel([0.362726, -1.263007, -2.645506, -0.803876, 1.570796, 1.933522],accel_mss,speed_ms,0,blend_radius_m)
    movel([0.362625, -1.263272, -2.645360, -0.803757, 1.570796, 1.933421],accel_mss,speed_ms,0,blend_radius_m)
    movel([0.362402, -1.263498, -2.645236, -0.803655, 1.570796, 1.933199],accel_mss,speed_ms,0,blend_radius_m)
    movel([0.361743, -1.263943, -2.644991, -0.803455, 1.570796, 1.932540],accel_mss,speed_ms,0,blend_radius_m)
    movel([0.361093, -1.264176, -2.644863, -0.803350, 1.570796, 1.931890],accel_mss,speed_ms,0,blend_radius_m)
    movel([0.359903, -1.264349, -2.644768, -0.803272, 1.570796, 1.930699],accel_mss,speed_ms,0,blend_radius_m)
    movel([0.358736, -1.264439, -2.644719, -0.803232, 1.570796, 1.929532],accel_mss,speed_ms,0,blend_radius_m)
    movel([0.358080, -1.264358, -2.644763, -0.803268, 1.570796, 1.928877],accel_mss,speed_ms,0,blend_radius_m)
    movel([0.357683, -1.264331, -2.644778, -0.803280, 1.570796, 1.928479],accel_mss,speed_ms,0,blend_radius_m)
    movel([0.357290, -1.264482, -2.644695, -0.803212, 1.570796, 1.928086],accel_mss,speed_ms,0,blend_radius_m)
    movel([0.357011, -1.264765, -2.644539, -0.803085, 1.570796, 1.927808],accel_mss,speed_ms,0,blend_radius_m)
    movel([0.356903, -1.265108, -2.644350, -0.802931, 1.570796, 1.927700],accel_mss,speed_ms,0,blend_radius_m)
    movel([0.357054, -1.265389, -2.644195, -0.802805, 1.570796, 1.927851],accel_mss,speed_ms,0,blend_radius_m)
    movel([0.357524, -1.265557, -2.644102, -0.802730, 1.570796, 1.928320],accel_mss,speed_ms,0,blend_radius_m)
    movel([0.358255, -1.265619, -2.644068, -0.802702, 1.570796, 1.929052],accel_mss,speed_ms,0,blend_radius_m)
    movel([0.359853, -1.265504, -2.644131, -0.802754, 1.570796, 1.930650],accel_mss,speed_ms,0,blend_radius_m)
    movel([0.360243, -1.265509, -2.644128, -0.802751, 1.570796, 1.931039],accel_mss,speed_ms,0,blend_radius_m)
    movel([0.360542, -1.265680, -2.644034, -0.802675, 1.570796, 1.931338],accel_mss,speed_ms,0,blend_radius_m)
    movel([0.360410, -1.266044, -2.643833, -0.802512, 1.570796, 1.931206],accel_mss,speed_ms,0,blend_radius_m)
    movel([0.360068, -1.266343, -2.643668, -0.802378, 1.570796, 1.930864],accel_mss,speed_ms,0,blend_radius_m)
    movel([0.358583, -1.266967, -2.643323, -0.802100, 1.570796, 1.929380],accel_mss,speed_ms,0,blend_radius_m)
    movel([0.356824, -1.267344, -2.643114, -0.801931, 1.570796, 1.927620],accel_mss,speed_ms,0,blend_radius_m)
    movel([0.356113, -1.267362, -2.643104, -0.801923, 1.570796, 1.926909],accel_mss,speed_ms,0,blend_radius_m)
    movel([0.354950, -1.267200, -2.643193, -0.801995, 1.570796, 1.925747],accel_mss,speed_ms,0,blend_radius_m)
    movel([0.354750, -1.267280, -2.643149, -0.801960, 1.570796, 1.925547],accel_mss,speed_ms,0,blend_radius_m)
    movel([0.354282, -1.267654, -2.642942, -0.801793, 1.570796, 1.925078],accel_mss,speed_ms,0,blend_radius_m)
    movel([0.354184, -1.267801, -2.642860, -0.801728, 1.570796, 1.924980],accel_mss,speed_ms,0,blend_radius_m)
    movel([0.354230, -1.268220, -2.642628, -0.801541, 1.570796, 1.925027],accel_mss,speed_ms,0,blend_radius_m)
    movel([0.354515, -1.268509, -2.642467, -0.801413, 1.570796, 1.925311],accel_mss,speed_ms,0,blend_radius_m)
    movel([0.355197, -1.268645, -2.642392, -0.801352, 1.570796, 1.925993],accel_mss,speed_ms,0,blend_radius_m)
    movel([0.356281, -1.268649, -2.642389, -0.801351, 1.570796, 1.927077],accel_mss,speed_ms,0,blend_radius_m)
    movel([0.358578, -1.268450, -2.642500, -0.801439, 1.570796, 1.929374],accel_mss,speed_ms,0,blend_radius_m)
    movel([0.358878, -1.268462, -2.642493, -0.801434, 1.570796, 1.929674],accel_mss,speed_ms,0,blend_radius_m)
    movel([0.358959, -1.268705, -2.642359, -0.801326, 1.570796, 1.929755],accel_mss,speed_ms,0,blend_radius_m)
    movel([0.358573, -1.269154, -2.642109, -0.801126, 1.570796, 1.929369],accel_mss,speed_ms,0,blend_radius_m)
    movel([0.357940, -1.269572, -2.641876, -0.800941, 1.570796, 1.928737],accel_mss,speed_ms,0,blend_radius_m)
    movel([0.357124, -1.269923, -2.641680, -0.800786, 1.570796, 1.927920],accel_mss,speed_ms,0,blend_radius_m)
    movel([0.355106, -1.270453, -2.641385, -0.800551, 1.570796, 1.925903],accel_mss,speed_ms,0,blend_radius_m)
    movel([0.354912, -1.270622, -2.641290, -0.800476, 1.570796, 1.925709],accel_mss,speed_ms,0,blend_radius_m)
    movel([0.354727, -1.271177, -2.640981, -0.800232, 1.570796, 1.925523],accel_mss,speed_ms,0,blend_radius_m)
    movel([0.354848, -1.271312, -2.640905, -0.800172, 1.570796, 1.925644],accel_mss,speed_ms,0,blend_radius_m)
    movel([0.357297, -1.271263, -2.640932, -0.800194, 1.570796, 1.928093],accel_mss,speed_ms,0,blend_radius_m)
    movel([0.357970, -1.271298, -2.640913, -0.800178, 1.570796, 1.928766],accel_mss,speed_ms,0,blend_radius_m)
    movel([0.359037, -1.271583, -2.640753, -0.800052, 1.570796, 1.929833],accel_mss,speed_ms,0,blend_radius_m)
    movel([0.359693, -1.271952, -2.640547, -0.799890, 1.570796, 1.930489],accel_mss,speed_ms,0,blend_radius_m)
    movel([0.360766, -1.272968, -2.639977, -0.799444, 1.570796, 1.931563],accel_mss,speed_ms,0,blend_radius_m)
    movel([0.360788, -1.273283, -2.639800, -0.799305, 1.570796, 1.931584],accel_mss,speed_ms,0,blend_radius_m)
    movel([0.360672, -1.273436, -2.639715, -0.799239, 1.570796, 1.931468],accel_mss,speed_ms,0,blend_radius_m)
    movel([0.360502, -1.273505, -2.639676, -0.799208, 1.570796, 1.931298],accel_mss,speed_ms,0,blend_radius_m)
    movel([0.359428, -1.273502, -2.639678, -0.799210, 1.570796, 1.930225],accel_mss,speed_ms,0,blend_radius_m)
    movel([0.358279, -1.273382, -2.639745, -0.799262, 1.570796, 1.929075],accel_mss,speed_ms,0,blend_radius_m)
    movel([0.356302, -1.272738, -2.640107, -0.799545, 1.570796, 1.927098],accel_mss,speed_ms,0,blend_radius_m)
    movel([0.355336, -1.273257, -2.639815, -0.799317, 1.570796, 1.926132],accel_mss,speed_ms,0,blend_radius_m)
    movel([0.354332, -1.273685, -2.639575, -0.799129, 1.570796, 1.925128],accel_mss,speed_ms,0,blend_radius_m)
    movel([0.353903, -1.273723, -2.639553, -0.799112, 1.570796, 1.924700],accel_mss,speed_ms,0,blend_radius_m)
    movel([0.351947, -1.273591, -2.639627, -0.799170, 1.570796, 1.922743],accel_mss,speed_ms,0,blend_radius_m)
    movel([0.351675, -1.273505, -2.639676, -0.799208, 1.570796, 1.922471],accel_mss,speed_ms,0,blend_radius_m)
    movel([0.351691, -1.273340, -2.639769, -0.799280, 1.570796, 1.922488],accel_mss,speed_ms,0,blend_radius_m)
    movel([0.352037, -1.272998, -2.639960, -0.799430, 1.570796, 1.922834],accel_mss,speed_ms,0,blend_radius_m)
    movel([0.352696, -1.272237, -2.640387, -0.799765, 1.570796, 1.923493],accel_mss,speed_ms,0,blend_radius_m)
    movel([0.352733, -1.271974, -2.640535, -0.799881, 1.570796, 1.923530],accel_mss,speed_ms,0,blend_radius_m)
    movel([0.352584, -1.271819, -2.640621, -0.799949, 1.570796, 1.923380],accel_mss,speed_ms,0,blend_radius_m)
    movel([0.352415, -1.271835, -2.640612, -0.799942, 1.570796, 1.923212],accel_mss,speed_ms,0,blend_radius_m)
    movel([0.351743, -1.272209, -2.640403, -0.799777, 1.570796, 1.922539],accel_mss,speed_ms,0,blend_radius_m)
    movel([0.351302, -1.272528, -2.640224, -0.799637, 1.570796, 1.922098],accel_mss,speed_ms,0,blend_radius_m)
    movel([0.350037, -1.273621, -2.639611, -0.799157, 1.570796, 1.920833],accel_mss,speed_ms,0,blend_radius_m)
    movel([0.349760, -1.273994, -2.639401, -0.798994, 1.570796, 1.920556],accel_mss,speed_ms,0,blend_radius_m)
    movel([0.349670, -1.274307, -2.639225, -0.798857, 1.570796, 1.920466],accel_mss,speed_ms,0,blend_radius_m)
    movel([0.349854, -1.274521, -2.639104, -0.798763, 1.570796, 1.920650],accel_mss,speed_ms,0,blend_radius_m)
    movel([0.351101, -1.274705, -2.639001, -0.798683, 1.570796, 1.921898],accel_mss,speed_ms,0,blend_radius_m)
    movel([0.352464, -1.274823, -2.638934, -0.798632, 1.570796, 1.923261],accel_mss,speed_ms,0,blend_radius_m)
    movel([0.354873, -1.274914, -2.638883, -0.798592, 1.570796, 1.925669],accel_mss,speed_ms,0,blend_radius_m)
    movel([0.355828, -1.275352, -2.638636, -0.798401, 1.570796, 1.926625],accel_mss,speed_ms,0,blend_radius_m)
    movel([0.356385, -1.276015, -2.638262, -0.798112, 1.570796, 1.927181],accel_mss,speed_ms,0,blend_radius_m)
    movel([0.356455, -1.276359, -2.638067, -0.797962, 1.570796, 1.927251],accel_mss,speed_ms,0,blend_radius_m)
    movel([0.356267, -1.276986, -2.637712, -0.797690, 1.570796, 1.927063],accel_mss,speed_ms,0,blend_radius_m)
    movel([0.356132, -1.277137, -2.637627, -0.797625, 1.570796, 1.926928],accel_mss,speed_ms,0,blend_radius_m)
    movel([0.355432, -1.277394, -2.637481, -0.797513, 1.570796, 1.926228],accel_mss,speed_ms,0,blend_radius_m)
    movel([0.355218, -1.277502, -2.637420, -0.797467, 1.570796, 1.926014],accel_mss,speed_ms,0,blend_radius_m)
    movel([0.354935, -1.277782, -2.637262, -0.797345, 1.570796, 1.925732],accel_mss,speed_ms,0,blend_radius_m)
    movel([0.354778, -1.278347, -2.636941, -0.797101, 1.570796, 1.925575],accel_mss,speed_ms,0,blend_radius_m)
    movel([0.355107, -1.280162, -2.635908, -0.796319, 1.570796, 1.925903],accel_mss,speed_ms,0,blend_radius_m)
    movel([0.355466, -1.280844, -2.635519, -0.796026, 1.570796, 1.926262],accel_mss,speed_ms,0,blend_radius_m)
    movel([0.355866, -1.281634, -2.635068, -0.795688, 1.570796, 1.926662],accel_mss,speed_ms,0,blend_radius_m)
    movel([0.355818, -1.282013, -2.634851, -0.795525, 1.570796, 1.926614],accel_mss,speed_ms,0,blend_radius_m)
    movel([0.355393, -1.283339, -2.634090, -0.794959, 1.570796, 1.926190],accel_mss,speed_ms,0,blend_radius_m)
    movel([0.355280, -1.283913, -2.633761, -0.794715, 1.570796, 1.926077],accel_mss,speed_ms,0,blend_radius_m)
    movel([0.355239, -1.287068, -2.631940, -0.793380, 1.570796, 1.926036],accel_mss,speed_ms,0,blend_radius_m)
    movel([0.355198, -1.287558, -2.631657, -0.793174, 1.570796, 1.925994],accel_mss,speed_ms,0,blend_radius_m)
    movel([0.354557, -1.290493, -2.629951, -0.791945, 1.570796, 1.925353],accel_mss,speed_ms,0,blend_radius_m)
    movel([0.354074, -1.292161, -2.628976, -0.791252, 1.570796, 1.924870],accel_mss,speed_ms,0,blend_radius_m)
    movel([0.353729, -1.292957, -2.628510, -0.790922, 1.570796, 1.924525],accel_mss,speed_ms,0,blend_radius_m)
    movel([0.353303, -1.293536, -2.628170, -0.790683, 1.570796, 1.924099],accel_mss,speed_ms,0,blend_radius_m)
    movel([0.352745, -1.294009, -2.627892, -0.790488, 1.570796, 1.923541],accel_mss,speed_ms,0,blend_radius_m)
    movel([0.352027, -1.294390, -2.627668, -0.790331, 1.570796, 1.922823],accel_mss,speed_ms,0,blend_radius_m)
    movel([0.351120, -1.294690, -2.627492, -0.790208, 1.570796, 1.921917],accel_mss,speed_ms,0,blend_radius_m)
    movel([0.350647, -1.294825, -2.627412, -0.790152, 1.570796, 1.921443],accel_mss,speed_ms,0,blend_radius_m)
    movel([0.349704, -1.295184, -2.627200, -0.790004, 1.570796, 1.920500],accel_mss,speed_ms,0,blend_radius_m)
    movel([0.349619, -1.295321, -2.627120, -0.789948, 1.570796, 1.920415],accel_mss,speed_ms,0,blend_radius_m)
    movel([0.349668, -1.296652, -2.626334, -0.789403, 1.570796, 1.920464],accel_mss,speed_ms,0,blend_radius_m)
    movel([0.349747, -1.297799, -2.625655, -0.788934, 1.570796, 1.920544],accel_mss,speed_ms,0,blend_radius_m)
    movel([0.349623, -1.298836, -2.625040, -0.788513, 1.570796, 1.920420],accel_mss,speed_ms,0,blend_radius_m)
    movel([0.349294, -1.299796, -2.624469, -0.788124, 1.570796, 1.920090],accel_mss,speed_ms,0,blend_radius_m)
    movel([0.348750, -1.300719, -2.623919, -0.787750, 1.570796, 1.919546],accel_mss,speed_ms,0,blend_radius_m)
    movel([0.348501, -1.301050, -2.623722, -0.787617, 1.570796, 1.919297],accel_mss,speed_ms,0,blend_radius_m)
    movel([0.347983, -1.301597, -2.623396, -0.787397, 1.570796, 1.918779],accel_mss,speed_ms,0,blend_radius_m)
    movel([0.347804, -1.301470, -2.623471, -0.787448, 1.570796, 1.918600],accel_mss,speed_ms,0,blend_radius_m)
    movel([0.347713, -1.300319, -2.624158, -0.787912, 1.570796, 1.918510],accel_mss,speed_ms,0,blend_radius_m)
    movel([0.347687, -1.299161, -2.624847, -0.788381, 1.570796, 1.918483],accel_mss,speed_ms,0,blend_radius_m)
    movel([0.347786, -1.298360, -2.625323, -0.788706, 1.570796, 1.918582],accel_mss,speed_ms,0,blend_radius_m)
    movel([0.347879, -1.297761, -2.625678, -0.788950, 1.570796, 1.918675],accel_mss,speed_ms,0,blend_radius_m)
    movel([0.347819, -1.297388, -2.625899, -0.789102, 1.570796, 1.918615],accel_mss,speed_ms,0,blend_radius_m)
    movel([0.347612, -1.297239, -2.625987, -0.789163, 1.570796, 1.918408],accel_mss,speed_ms,0,blend_radius_m)
    movel([0.347120, -1.297347, -2.625923, -0.789119, 1.570796, 1.917916],accel_mss,speed_ms,0,blend_radius_m)
    movel([0.347627, -1.296370, -2.626501, -0.789518, 1.570796, 1.918423],accel_mss,speed_ms,0,blend_radius_m)
    movel([0.348523, -1.294312, -2.627714, -0.790363, 1.570796, 1.919320],accel_mss,speed_ms,0,blend_radius_m)
    movel([0.350665, -1.288938, -2.630856, -0.792595, 1.570796, 1.921461],accel_mss,speed_ms,0,blend_radius_m)
    movel([0.352150, -1.285018, -2.633125, -0.794246, 1.570796, 1.922946],accel_mss,speed_ms,0,blend_radius_m)
    movel([0.351819, -1.284510, -2.633417, -0.794462, 1.570796, 1.922616],accel_mss,speed_ms,0,blend_radius_m)
    movel([0.351434, -1.284122, -2.633640, -0.794626, 1.570796, 1.922231],accel_mss,speed_ms,0,blend_radius_m)
    movel([0.350820, -1.283802, -2.633824, -0.794762, 1.570796, 1.921617],accel_mss,speed_ms,0,blend_radius_m)
    movel([0.350172, -1.283609, -2.633936, -0.794845, 1.570796, 1.920969],accel_mss,speed_ms,0,blend_radius_m)
    movel([0.349723, -1.283675, -2.633897, -0.794816, 1.570796, 1.920519],accel_mss,speed_ms,0,blend_radius_m)
    movel([0.349384, -1.283933, -2.633749, -0.794707, 1.570796, 1.920180],accel_mss,speed_ms,0,blend_radius_m)
    movel([0.349259, -1.284255, -2.633564, -0.794570, 1.570796, 1.920055],accel_mss,speed_ms,0,blend_radius_m)
    movel([0.349406, -1.284586, -2.633374, -0.794429, 1.570796, 1.920202],accel_mss,speed_ms,0,blend_radius_m)
    movel([0.349805, -1.284839, -2.633228, -0.794322, 1.570796, 1.920602],accel_mss,speed_ms,0,blend_radius_m)
    movel([0.350545, -1.285322, -2.632949, -0.794117, 1.570796, 1.921341],accel_mss,speed_ms,0,blend_radius_m)
    movel([0.350697, -1.285597, -2.632791, -0.794001, 1.570796, 1.921493],accel_mss,speed_ms,0,blend_radius_m)
    movel([0.350707, -1.285952, -2.632586, -0.793851, 1.570796, 1.921503],accel_mss,speed_ms,0,blend_radius_m)
    movel([0.350365, -1.287144, -2.631897, -0.793348, 1.570796, 1.921161],accel_mss,speed_ms,0,blend_radius_m)
    movel([0.348730, -1.291198, -2.629539, -0.791652, 1.570796, 1.919526],accel_mss,speed_ms,0,blend_radius_m)
    movel([0.346425, -1.296587, -2.626373, -0.789429, 1.570796, 1.917222],accel_mss,speed_ms,0,blend_radius_m)
    movel([0.346185, -1.296972, -2.626145, -0.789272, 1.570796, 1.916981],accel_mss,speed_ms,0,blend_radius_m)
    movel([0.345850, -1.297284, -2.625960, -0.789144, 1.570796, 1.916646],accel_mss,speed_ms,0,blend_radius_m)
    movel([0.345486, -1.297450, -2.625862, -0.789077, 1.570796, 1.916282],accel_mss,speed_ms,0,blend_radius_m)
    movel([0.343358, -1.297485, -2.625841, -0.789062, 1.570796, 1.914154],accel_mss,speed_ms,0,blend_radius_m)
    movel([0.342997, -1.297586, -2.625782, -0.789021, 1.570796, 1.913793],accel_mss,speed_ms,0,blend_radius_m)
    movel([0.341689, -1.298489, -2.625246, -0.788654, 1.570796, 1.912486],accel_mss,speed_ms,0,blend_radius_m)
    movel([0.340503, -1.299311, -2.624758, -0.788320, 1.570796, 1.911299],accel_mss,speed_ms,0,blend_radius_m)
    movel([0.339513, -1.299812, -2.624460, -0.788117, 1.570796, 1.910309],accel_mss,speed_ms,0,blend_radius_m)
    movel([0.338596, -1.300046, -2.624320, -0.788022, 1.570796, 1.909392],accel_mss,speed_ms,0,blend_radius_m)
    movel([0.337637, -1.300060, -2.624312, -0.788017, 1.570796, 1.908433],accel_mss,speed_ms,0,blend_radius_m)
    movel([0.337255, -1.299999, -2.624349, -0.788042, 1.570796, 1.908051],accel_mss,speed_ms,0,blend_radius_m)
    movel([0.336287, -1.299626, -2.624571, -0.788193, 1.570796, 1.907083],accel_mss,speed_ms,0,blend_radius_m)
    movel([0.335954, -1.299452, -2.624674, -0.788263, 1.570796, 1.906750],accel_mss,speed_ms,0,blend_radius_m)
    movel([0.335607, -1.299452, -2.624674, -0.788263, 1.570796, 1.906404],accel_mss,speed_ms,0,blend_radius_m)
    movel([0.335283, -1.299618, -2.624576, -0.788196, 1.570796, 1.906079],accel_mss,speed_ms,0,blend_radius_m)
    movel([0.334995, -1.299928, -2.624391, -0.788070, 1.570796, 1.905791],accel_mss,speed_ms,0,blend_radius_m)
    movel([0.334978, -1.300240, -2.624205, -0.787944, 1.570796, 1.905774],accel_mss,speed_ms,0,blend_radius_m)
    movel([0.335512, -1.300652, -2.623959, -0.787777, 1.570796, 1.906309],accel_mss,speed_ms,0,blend_radius_m)
    movel([0.336228, -1.301005, -2.623749, -0.787635, 1.570796, 1.907024],accel_mss,speed_ms,0,blend_radius_m)
    movel([0.336964, -1.301171, -2.623650, -0.787568, 1.570796, 1.907760],accel_mss,speed_ms,0,blend_radius_m)
    movel([0.338179, -1.301133, -2.623672, -0.787583, 1.570796, 1.908975],accel_mss,speed_ms,0,blend_radius_m)
    movel([0.339489, -1.300792, -2.623876, -0.787721, 1.570796, 1.910285],accel_mss,speed_ms,0,blend_radius_m)
    movel([0.340829, -1.300161, -2.624252, -0.787976, 1.570796, 1.911625],accel_mss,speed_ms,0,blend_radius_m)
    movel([0.342999, -1.298670, -2.625139, -0.788580, 1.570796, 1.913795],accel_mss,speed_ms,0,blend_radius_m)
    movel([0.343285, -1.298580, -2.625192, -0.788617, 1.570796, 1.914081],accel_mss,speed_ms,0,blend_radius_m)
    movel([0.345336, -1.298633, -2.625161, -0.788595, 1.570796, 1.916132],accel_mss,speed_ms,0,blend_radius_m)
    movel([0.345760, -1.298481, -2.625251, -0.788657, 1.570796, 1.916556],accel_mss,speed_ms,0,blend_radius_m)
    movel([0.346208, -1.298168, -2.625437, -0.788784, 1.570796, 1.917004],accel_mss,speed_ms,0,blend_radius_m)
    movel([0.346803, -1.297652, -2.625742, -0.788994, 1.570796, 1.917599],accel_mss,speed_ms,0,blend_radius_m)
    movel([0.346537, -1.299846, -2.624440, -0.788103, 1.570796, 1.917333],accel_mss,speed_ms,0,blend_radius_m)
    movel([0.346609, -1.301127, -2.623676, -0.787586, 1.570796, 1.917406],accel_mss,speed_ms,0,blend_radius_m)
    movel([0.347204, -1.304153, -2.621864, -0.786372, 1.570796, 1.918000],accel_mss,speed_ms,0,blend_radius_m)
    movel([0.347600, -1.305730, -2.620915, -0.785744, 1.570796, 1.918397],accel_mss,speed_ms,0,blend_radius_m)
    movel([0.347852, -1.307513, -2.619838, -0.785038, 1.570796, 1.918648],accel_mss,speed_ms,0,blend_radius_m)
    movel([0.347751, -1.308045, -2.619516, -0.784829, 1.570796, 1.918548],accel_mss,speed_ms,0,blend_radius_m)
    movel([0.347558, -1.308437, -2.619278, -0.784674, 1.570796, 1.918354],accel_mss,speed_ms,0,blend_radius_m)
    movel([0.347131, -1.308272, -2.619378, -0.784739, 1.570796, 1.917927],accel_mss,speed_ms,0,blend_radius_m)
    movel([0.346978, -1.308275, -2.619376, -0.784738, 1.570796, 1.917775],accel_mss,speed_ms,0,blend_radius_m)
    movel([0.346645, -1.308445, -2.619273, -0.784671, 1.570796, 1.917441],accel_mss,speed_ms,0,blend_radius_m)
    movel([0.346491, -1.308650, -2.619149, -0.784590, 1.570796, 1.917287],accel_mss,speed_ms,0,blend_radius_m)
    movel([0.345986, -1.310277, -2.618160, -0.783952, 1.570796, 1.916782],accel_mss,speed_ms,0,blend_radius_m)
    movel([0.345941, -1.310875, -2.617796, -0.783719, 1.570796, 1.916738],accel_mss,speed_ms,0,blend_radius_m)
    movel([0.346571, -1.314946, -2.615303, -0.782140, 1.570796, 1.917368],accel_mss,speed_ms,0,blend_radius_m)
    movel([0.346668, -1.317033, -2.614017, -0.781340, 1.570796, 1.917464],accel_mss,speed_ms,0,blend_radius_m)
    movel([0.346570, -1.318742, -2.612959, -0.780688, 1.570796, 1.917367],accel_mss,speed_ms,0,blend_radius_m)
    movel([0.346433, -1.318987, -2.612807, -0.780595, 1.570796, 1.917230],accel_mss,speed_ms,0,blend_radius_m)
    movel([0.346169, -1.319118, -2.612726, -0.780545, 1.570796, 1.916965],accel_mss,speed_ms,0,blend_radius_m)
    movel([0.345914, -1.318263, -2.613256, -0.780870, 1.570796, 1.916710],accel_mss,speed_ms,0,blend_radius_m)
    movel([0.345834, -1.318084, -2.613367, -0.780939, 1.570796, 1.916630],accel_mss,speed_ms,0,blend_radius_m)
    movel([0.345538, -1.317964, -2.613441, -0.780984, 1.570796, 1.916334],accel_mss,speed_ms,0,blend_radius_m)
    movel([0.345163, -1.318113, -2.613348, -0.780927, 1.570796, 1.915960],accel_mss,speed_ms,0,blend_radius_m)
    movel([0.344928, -1.318407, -2.613167, -0.780816, 1.570796, 1.915724],accel_mss,speed_ms,0,blend_radius_m)
    movel([0.344837, -1.318926, -2.612845, -0.780618, 1.570796, 1.915633],accel_mss,speed_ms,0,blend_radius_m)
    movel([0.344887, -1.319792, -2.612307, -0.780290, 1.570796, 1.915683],accel_mss,speed_ms,0,blend_radius_m)
    movel([0.345424, -1.322665, -2.610516, -0.779208, 1.570796, 1.916220],accel_mss,speed_ms,0,blend_radius_m)
    movel([0.345851, -1.323939, -2.609718, -0.778732, 1.570796, 1.916647],accel_mss,speed_ms,0,blend_radius_m)
    movel([0.346396, -1.325138, -2.608965, -0.778285, 1.570796, 1.917192],accel_mss,speed_ms,0,blend_radius_m)
    movel([0.347861, -1.327323, -2.607589, -0.777477, 1.570796, 1.918658],accel_mss,speed_ms,0,blend_radius_m)
    movel([0.349869, -1.329335, -2.606316, -0.776738, 1.570796, 1.920665],accel_mss,speed_ms,0,blend_radius_m)
    movel([0.351898, -1.331280, -2.605080, -0.776029, 1.570796, 1.922694],accel_mss,speed_ms,0,blend_radius_m)
    movel([0.352340, -1.331875, -2.604700, -0.775814, 1.570796, 1.923136],accel_mss,speed_ms,0,blend_radius_m)
    movel([0.350918, -1.332006, -2.604617, -0.775766, 1.570796, 1.921714],accel_mss,speed_ms,0,blend_radius_m)
    movel([0.349891, -1.331836, -2.604725, -0.775828, 1.570796, 1.920687],accel_mss,speed_ms,0,blend_radius_m)
    movel([0.347985, -1.331207, -2.605126, -0.776056, 1.570796, 1.918781],accel_mss,speed_ms,0,blend_radius_m)
    movel([0.347410, -1.330790, -2.605392, -0.776208, 1.570796, 1.918207],accel_mss,speed_ms,0,blend_radius_m)
    movel([0.346904, -1.330134, -2.605809, -0.776447, 1.570796, 1.917700],accel_mss,speed_ms,0,blend_radius_m)
    movel([0.346458, -1.329245, -2.606373, -0.776771, 1.570796, 1.917254],accel_mss,speed_ms,0,blend_radius_m)
    movel([0.345898, -1.327568, -2.607434, -0.777387, 1.570796, 1.916694],accel_mss,speed_ms,0,blend_radius_m)
    movel([0.345725, -1.327201, -2.607666, -0.777522, 1.570796, 1.916522],accel_mss,speed_ms,0,blend_radius_m)
    movel([0.345380, -1.326926, -2.607840, -0.777623, 1.570796, 1.916176],accel_mss,speed_ms,0,blend_radius_m)
    movel([0.345140, -1.327015, -2.607784, -0.777591, 1.570796, 1.915936],accel_mss,speed_ms,0,blend_radius_m)
    movel([0.344946, -1.327204, -2.607664, -0.777521, 1.570796, 1.915742],accel_mss,speed_ms,0,blend_radius_m)
    movel([0.344757, -1.327759, -2.607313, -0.777316, 1.570796, 1.915553],accel_mss,speed_ms,0,blend_radius_m)
    movel([0.344908, -1.328691, -2.606724, -0.776974, 1.570796, 1.915704],accel_mss,speed_ms,0,blend_radius_m)
    movel([0.345419, -1.330038, -2.605870, -0.776482, 1.570796, 1.916215],accel_mss,speed_ms,0,blend_radius_m)
    movel([0.345797, -1.331066, -2.605216, -0.776107, 1.570796, 1.916593],accel_mss,speed_ms,0,blend_radius_m)
    movel([0.348345, -1.334794, -2.602833, -0.774762, 1.570796, 1.919141],accel_mss,speed_ms,0,blend_radius_m)
    movel([0.348348, -1.334943, -2.602738, -0.774708, 1.570796, 1.919144],accel_mss,speed_ms,0,blend_radius_m)
    movel([0.348235, -1.335071, -2.602656, -0.774662, 1.570796, 1.919031],accel_mss,speed_ms,0,blend_radius_m)
    movel([0.348091, -1.335095, -2.602640, -0.774654, 1.570796, 1.918887],accel_mss,speed_ms,0,blend_radius_m)
    movel([0.347482, -1.334786, -2.602838, -0.774764, 1.570796, 1.918278],accel_mss,speed_ms,0,blend_radius_m)
    movel([0.346831, -1.334254, -2.603179, -0.774955, 1.570796, 1.917627],accel_mss,speed_ms,0,blend_radius_m)
    movel([0.346133, -1.333276, -2.603806, -0.775307, 1.570796, 1.916929],accel_mss,speed_ms,0,blend_radius_m)
    movel([0.345920, -1.333038, -2.603958, -0.775393, 1.570796, 1.916716],accel_mss,speed_ms,0,blend_radius_m)
    movel([0.345535, -1.332899, -2.604047, -0.775443, 1.570796, 1.916331],accel_mss,speed_ms,0,blend_radius_m)
    movel([0.345186, -1.333102, -2.603917, -0.775370, 1.570796, 1.915982],accel_mss,speed_ms,0,blend_radius_m)
    movel([0.345021, -1.333413, -2.603718, -0.775258, 1.570796, 1.915817],accel_mss,speed_ms,0,blend_radius_m)
    movel([0.345083, -1.333884, -2.603417, -0.775088, 1.570796, 1.915879],accel_mss,speed_ms,0,blend_radius_m)
    movel([0.345399, -1.334578, -2.602972, -0.774839, 1.570796, 1.916195],accel_mss,speed_ms,0,blend_radius_m)
    movel([0.346092, -1.335659, -2.602278, -0.774452, 1.570796, 1.916888],accel_mss,speed_ms,0,blend_radius_m)
    movel([0.346945, -1.336588, -2.601680, -0.774121, 1.570796, 1.917741],accel_mss,speed_ms,0,blend_radius_m)
    movel([0.348024, -1.337418, -2.601145, -0.773826, 1.570796, 1.918820],accel_mss,speed_ms,0,blend_radius_m)
    movel([0.349390, -1.338207, -2.600635, -0.773546, 1.570796, 1.920186],accel_mss,speed_ms,0,blend_radius_m)
    movel([0.350690, -1.338898, -2.600189, -0.773302, 1.570796, 1.921486],accel_mss,speed_ms,0,blend_radius_m)
    movel([0.351660, -1.339676, -2.599685, -0.773028, 1.570796, 1.922457],accel_mss,speed_ms,0,blend_radius_m)
    movel([0.351587, -1.339943, -2.599511, -0.772934, 1.570796, 1.922383],accel_mss,speed_ms,0,blend_radius_m)
    movel([0.351201, -1.340150, -2.599377, -0.772862, 1.570796, 1.921997],accel_mss,speed_ms,0,blend_radius_m)
    movel([0.350068, -1.340251, -2.599312, -0.772826, 1.570796, 1.920865],accel_mss,speed_ms,0,blend_radius_m)
    movel([0.347733, -1.340175, -2.599361, -0.772853, 1.570796, 1.918529],accel_mss,speed_ms,0,blend_radius_m)
    movel([0.346067, -1.339737, -2.599645, -0.773007, 1.570796, 1.916864],accel_mss,speed_ms,0,blend_radius_m)
    movel([0.344058, -1.338814, -2.600243, -0.773332, 1.570796, 1.914854],accel_mss,speed_ms,0,blend_radius_m)
    movel([0.342043, -1.337608, -2.601022, -0.773759, 1.570796, 1.912839],accel_mss,speed_ms,0,blend_radius_m)
    movel([0.340318, -1.336274, -2.601882, -0.774233, 1.570796, 1.911114],accel_mss,speed_ms,0,blend_radius_m)
    movel([0.339385, -1.335196, -2.602575, -0.774618, 1.570796, 1.910182],accel_mss,speed_ms,0,blend_radius_m)
    movel([0.338949, -1.334047, -2.603312, -0.775030, 1.570796, 1.909745],accel_mss,speed_ms,0,blend_radius_m)
    movel([0.338888, -1.332376, -2.604381, -0.775632, 1.570796, 1.909685],accel_mss,speed_ms,0,blend_radius_m)
    movel([0.339669, -1.325128, -2.608972, -0.778289, 1.570796, 1.910465],accel_mss,speed_ms,0,blend_radius_m)
    movel([0.339816, -1.322562, -2.610581, -0.779247, 1.570796, 1.910613],accel_mss,speed_ms,0,blend_radius_m)
    movel([0.339702, -1.320892, -2.611623, -0.779875, 1.570796, 1.910498],accel_mss,speed_ms,0,blend_radius_m)
    movel([0.339292, -1.319812, -2.612295, -0.780283, 1.570796, 1.910089],accel_mss,speed_ms,0,blend_radius_m)
    movel([0.338974, -1.319382, -2.612561, -0.780445, 1.570796, 1.909771],accel_mss,speed_ms,0,blend_radius_m)
    movel([0.338744, -1.319222, -2.612661, -0.780506, 1.570796, 1.909540],accel_mss,speed_ms,0,blend_radius_m)
    movel([0.337839, -1.319260, -2.612637, -0.780492, 1.570796, 1.908636],accel_mss,speed_ms,0,blend_radius_m)
    movel([0.336867, -1.319419, -2.612539, -0.780431, 1.570796, 1.907663],accel_mss,speed_ms,0,blend_radius_m)
    movel([0.339841, -1.312506, -2.616799, -0.783083, 1.570796, 1.910637],accel_mss,speed_ms,0,blend_radius_m)
    movel([0.340523, -1.310356, -2.618112, -0.783921, 1.570796, 1.911319],accel_mss,speed_ms,0,blend_radius_m)
    movel([0.341098, -1.307995, -2.619546, -0.784848, 1.570796, 1.911895],accel_mss,speed_ms,0,blend_radius_m)
    movel([0.341564, -1.305435, -2.621092, -0.785861, 1.570796, 1.912360],accel_mss,speed_ms,0,blend_radius_m)
    movel([0.342069, -1.301474, -2.623469, -0.787446, 1.570796, 1.912866],accel_mss,speed_ms,0,blend_radius_m)
    movel([0.342031, -1.300709, -2.623925, -0.787754, 1.570796, 1.912827],accel_mss,speed_ms,0,blend_radius_m)
    movel([0.341772, -1.300496, -2.624052, -0.787840, 1.570796, 1.912568],accel_mss,speed_ms,0,blend_radius_m)
    movel([0.341611, -1.300511, -2.624044, -0.787834, 1.570796, 1.912407],accel_mss,speed_ms,0,blend_radius_m)
    movel([0.341193, -1.300754, -2.623898, -0.787736, 1.570796, 1.911989],accel_mss,speed_ms,0,blend_radius_m)
    movel([0.341108, -1.300942, -2.623786, -0.787661, 1.570796, 1.911904],accel_mss,speed_ms,0,blend_radius_m)
    movel([0.340769, -1.303157, -2.622462, -0.786770, 1.570796, 1.911565],accel_mss,speed_ms,0,blend_radius_m)
    movel([0.340282, -1.306746, -2.620301, -0.785341, 1.570796, 1.911078],accel_mss,speed_ms,0,blend_radius_m)
    movel([0.339658, -1.309679, -2.618524, -0.784186, 1.570796, 1.910454],accel_mss,speed_ms,0,blend_radius_m)
    movel([0.338789, -1.312407, -2.616860, -0.783122, 1.570796, 1.909585],accel_mss,speed_ms,0,blend_radius_m)
    movel([0.336594, -1.317561, -2.613690, -0.781138, 1.570796, 1.907390],accel_mss,speed_ms,0,blend_radius_m)
    movel([0.335965, -1.319263, -2.612636, -0.780491, 1.570796, 1.906761],accel_mss,speed_ms,0,blend_radius_m)
    movel([0.335642, -1.320479, -2.611880, -0.780030, 1.570796, 1.906438],accel_mss,speed_ms,0,blend_radius_m)
    movel([0.335645, -1.320745, -2.611714, -0.779930, 1.570796, 1.906441],accel_mss,speed_ms,0,blend_radius_m)
    movel([0.335924, -1.321010, -2.611549, -0.779830, 1.570796, 1.906721],accel_mss,speed_ms,0,blend_radius_m)
    movel([0.336103, -1.320992, -2.611560, -0.779837, 1.570796, 1.906899],accel_mss,speed_ms,0,blend_radius_m)
    movel([0.337252, -1.320303, -2.611989, -0.780097, 1.570796, 1.908048],accel_mss,speed_ms,0,blend_radius_m)
    movel([0.337507, -1.320188, -2.612061, -0.780140, 1.570796, 1.908303],accel_mss,speed_ms,0,blend_radius_m)
    movel([0.337950, -1.320269, -2.612011, -0.780110, 1.570796, 1.908746],accel_mss,speed_ms,0,blend_radius_m)
    movel([0.338105, -1.320393, -2.611933, -0.780063, 1.570796, 1.908901],accel_mss,speed_ms,0,blend_radius_m)
    movel([0.338499, -1.321148, -2.611463, -0.779778, 1.570796, 1.909296],accel_mss,speed_ms,0,blend_radius_m)
    movel([0.338619, -1.322079, -2.610882, -0.779428, 1.570796, 1.909415],accel_mss,speed_ms,0,blend_radius_m)
    movel([0.338607, -1.323734, -2.609847, -0.778808, 1.570796, 1.909403],accel_mss,speed_ms,0,blend_radius_m)
    movel([0.338497, -1.325713, -2.608604, -0.778072, 1.570796, 1.909293],accel_mss,speed_ms,0,blend_radius_m)
    movel([0.337825, -1.331760, -2.604774, -0.775855, 1.570796, 1.908621],accel_mss,speed_ms,0,blend_radius_m)
    movel([0.337729, -1.333960, -2.603368, -0.775061, 1.570796, 1.908525],accel_mss,speed_ms,0,blend_radius_m)
    movel([0.337828, -1.334753, -2.602860, -0.774776, 1.570796, 1.908625],accel_mss,speed_ms,0,blend_radius_m)
    movel([0.338065, -1.335471, -2.602398, -0.774519, 1.570796, 1.908862],accel_mss,speed_ms,0,blend_radius_m)
    movel([0.338454, -1.336152, -2.601961, -0.774276, 1.570796, 1.909250],accel_mss,speed_ms,0,blend_radius_m)
    movel([0.338964, -1.336741, -2.601582, -0.774067, 1.570796, 1.909760],accel_mss,speed_ms,0,blend_radius_m)
    movel([0.340712, -1.338194, -2.600644, -0.773551, 1.570796, 1.911508],accel_mss,speed_ms,0,blend_radius_m)
    movel([0.342899, -1.339625, -2.599718, -0.773046, 1.570796, 1.913696],accel_mss,speed_ms,0,blend_radius_m)
    movel([0.344890, -1.340572, -2.599103, -0.772714, 1.570796, 1.915686],accel_mss,speed_ms,0,blend_radius_m)
    movel([0.346845, -1.341109, -2.598754, -0.772526, 1.570796, 1.917641],accel_mss,speed_ms,0,blend_radius_m)
    movel([0.348910, -1.341292, -2.598636, -0.772462, 1.570796, 1.919706],accel_mss,speed_ms,0,blend_radius_m)
    movel([0.349916, -1.341238, -2.598671, -0.772481, 1.570796, 1.920712],accel_mss,speed_ms,0,blend_radius_m)
    movel([0.350844, -1.341075, -2.598776, -0.772537, 1.570796, 1.921641],accel_mss,speed_ms,0,blend_radius_m)
    movel([0.351639, -1.340823, -2.598940, -0.772626, 1.570796, 1.922435],accel_mss,speed_ms,0,blend_radius_m)
    movel([0.352216, -1.340492, -2.599155, -0.772742, 1.570796, 1.923012],accel_mss,speed_ms,0,blend_radius_m)
    movel([0.352535, -1.340162, -2.599370, -0.772858, 1.570796, 1.923331],accel_mss,speed_ms,0,blend_radius_m)
    movel([0.352711, -1.339788, -2.599612, -0.772989, 1.570796, 1.923508],accel_mss,speed_ms,0,blend_radius_m)
    movel([0.352670, -1.338983, -2.600134, -0.773272, 1.570796, 1.923466],accel_mss,speed_ms,0,blend_radius_m)
    movel([0.352283, -1.338499, -2.600447, -0.773443, 1.570796, 1.923079],accel_mss,speed_ms,0,blend_radius_m)
    speed_ms = 0.005
    movel([0.352283, -1.329519, -2.596260, -0.786610, 1.570796, 1.923079],accel_mss,speed_ms,0,blend_radius_m)
    speed_ms = 0.040
    movel([0.376692, -1.289857, -2.620534, -0.801998, 1.570796, 1.947489],accel_mss,speed_ms,0,blend_radius_m)
    speed_ms = 0.005
    movel([0.376692, -1.299076, -2.624898, -0.788415, 1.570796, 1.947489],accel_mss,speed_ms,0,blend_radius_m)
    speed_ms = 0.025
    movel([0.376336, -1.299185, -2.624833, -0.788371, 1.570796, 1.947133],accel_mss,speed_ms,0,blend_radius_m)
    movel([0.376131, -1.299097, -2.624885, -0.788407, 1.570796, 1.946927],accel_mss,speed_ms,0,blend_radius_m)
    movel([0.376054, -1.298763, -2.625084, -0.788543, 1.570796, 1.946850],accel_mss,speed_ms,0,blend_radius_m)
    movel([0.376104, -1.298048, -2.625508, -0.788833, 1.570796, 1.946900],accel_mss,speed_ms,0,blend_radius_m)
    movel([0.376058, -1.296778, -2.626260, -0.789351, 1.570796, 1.946854],accel_mss,speed_ms,0,blend_radius_m)
    movel([0.375637, -1.295710, -2.626891, -0.789789, 1.570796, 1.946434],accel_mss,speed_ms,0,blend_radius_m)
    movel([0.374832, -1.294850, -2.627397, -0.790142, 1.570796, 1.945629],accel_mss,speed_ms,0,blend_radius_m)
    movel([0.373646, -1.294203, -2.627778, -0.790408, 1.570796, 1.944442],accel_mss,speed_ms,0,blend_radius_m)
    movel([0.372552, -1.293986, -2.627906, -0.790497, 1.570796, 1.943349],accel_mss,speed_ms,0,blend_radius_m)
    movel([0.371758, -1.293997, -2.627899, -0.790493, 1.570796, 1.942554],accel_mss,speed_ms,0,blend_radius_m)
    movel([0.368930, -1.294253, -2.627749, -0.790387, 1.570796, 1.939726],accel_mss,speed_ms,0,blend_radius_m)
    movel([0.367884, -1.294435, -2.627642, -0.790312, 1.570796, 1.938680],accel_mss,speed_ms,0,blend_radius_m)
    movel([0.361981, -1.296203, -2.626600, -0.789587, 1.570796, 1.932777],accel_mss,speed_ms,0,blend_radius_m)
    movel([0.360166, -1.296588, -2.626372, -0.789429, 1.570796, 1.930963],accel_mss,speed_ms,0,blend_radius_m)
    movel([0.358903, -1.296613, -2.626357, -0.789419, 1.570796, 1.929699],accel_mss,speed_ms,0,blend_radius_m)
    movel([0.357969, -1.296301, -2.626542, -0.789546, 1.570796, 1.928765],accel_mss,speed_ms,0,blend_radius_m)
    movel([0.357354, -1.295765, -2.626858, -0.789766, 1.570796, 1.928151],accel_mss,speed_ms,0,blend_radius_m)
    movel([0.356857, -1.295008, -2.627305, -0.790077, 1.570796, 1.927653],accel_mss,speed_ms,0,blend_radius_m)
    movel([0.356491, -1.294056, -2.627865, -0.790469, 1.570796, 1.927288],accel_mss,speed_ms,0,blend_radius_m)
    movel([0.356273, -1.292935, -2.628523, -0.790932, 1.570796, 1.927070],accel_mss,speed_ms,0,blend_radius_m)
    movel([0.356136, -1.291337, -2.629458, -0.791594, 1.570796, 1.926932],accel_mss,speed_ms,0,blend_radius_m)
    movel([0.356197, -1.290204, -2.630119, -0.792066, 1.570796, 1.926994],accel_mss,speed_ms,0,blend_radius_m)
    movel([0.356442, -1.289402, -2.630586, -0.792401, 1.570796, 1.927239],accel_mss,speed_ms,0,blend_radius_m)
    movel([0.356625, -1.289115, -2.630753, -0.792521, 1.570796, 1.927421],accel_mss,speed_ms,0,blend_radius_m)
    movel([0.356891, -1.288871, -2.630895, -0.792623, 1.570796, 1.927687],accel_mss,speed_ms,0,blend_radius_m)
    movel([0.357271, -1.288699, -2.630995, -0.792695, 1.570796, 1.928068],accel_mss,speed_ms,0,blend_radius_m)
    movel([0.357509, -1.288775, -2.630951, -0.792663, 1.570796, 1.928306],accel_mss,speed_ms,0,blend_radius_m)
    movel([0.357591, -1.289153, -2.630731, -0.792505, 1.570796, 1.928388],accel_mss,speed_ms,0,blend_radius_m)
    movel([0.357503, -1.291105, -2.629593, -0.791690, 1.570796, 1.928300],accel_mss,speed_ms,0,blend_radius_m)
    movel([0.357916, -1.292037, -2.629049, -0.791303, 1.570796, 1.928712],accel_mss,speed_ms,0,blend_radius_m)
    movel([0.358789, -1.292745, -2.628634, -0.791010, 1.570796, 1.929586],accel_mss,speed_ms,0,blend_radius_m)
    movel([0.360174, -1.293277, -2.628322, -0.790790, 1.570796, 1.930970],accel_mss,speed_ms,0,blend_radius_m)
    movel([0.361376, -1.293439, -2.628227, -0.790723, 1.570796, 1.932172],accel_mss,speed_ms,0,blend_radius_m)
    movel([0.362843, -1.293333, -2.628289, -0.790767, 1.570796, 1.933639],accel_mss,speed_ms,0,blend_radius_m)
    movel([0.364580, -1.292966, -2.628505, -0.790919, 1.570796, 1.935377],accel_mss,speed_ms,0,blend_radius_m)
    movel([0.366612, -1.292326, -2.628879, -0.791184, 1.570796, 1.937409],accel_mss,speed_ms,0,blend_radius_m)
    movel([0.369354, -1.291461, -2.629385, -0.791542, 1.570796, 1.940150],accel_mss,speed_ms,0,blend_radius_m)
    movel([0.371348, -1.291100, -2.629596, -0.791692, 1.570796, 1.942144],accel_mss,speed_ms,0,blend_radius_m)
    movel([0.372960, -1.291182, -2.629549, -0.791659, 1.570796, 1.943756],accel_mss,speed_ms,0,blend_radius_m)
    movel([0.374478, -1.291691, -2.629251, -0.791447, 1.570796, 1.945274],accel_mss,speed_ms,0,blend_radius_m)
    movel([0.375306, -1.292251, -2.628923, -0.791215, 1.570796, 1.946102],accel_mss,speed_ms,0,blend_radius_m)
    movel([0.376112, -1.293129, -2.628409, -0.790851, 1.570796, 1.946908],accel_mss,speed_ms,0,blend_radius_m)
    movel([0.376774, -1.294142, -2.627814, -0.790433, 1.570796, 1.947571],accel_mss,speed_ms,0,blend_radius_m)
    movel([0.377159, -1.295136, -2.627229, -0.790024, 1.570796, 1.947955],accel_mss,speed_ms,0,blend_radius_m)
    movel([0.377326, -1.296999, -2.626129, -0.789261, 1.570796, 1.948122],accel_mss,speed_ms,0,blend_radius_m)
    movel([0.377303, -1.298077, -2.625490, -0.788821, 1.570796, 1.948099],accel_mss,speed_ms,0,blend_radius_m)
    movel([0.377116, -1.298750, -2.625092, -0.788548, 1.570796, 1.947912],accel_mss,speed_ms,0,blend_radius_m)
    movel([0.377000, -1.298867, -2.625022, -0.788500, 1.570796, 1.947796],accel_mss,speed_ms,0,blend_radius_m)
    movel([0.376692, -1.299076, -2.624898, -0.788415, 1.570796, 1.947489],accel_mss,speed_ms,0,blend_radius_m)
    movel([0.376336, -1.299185, -2.624833, -0.788371, 1.570796, 1.947133],accel_mss,speed_ms,0,blend_radius_m)
    movel([0.376131, -1.299097, -2.624885, -0.788407, 1.570796, 1.946927],accel_mss,speed_ms,0,blend_radius_m)
    movel([0.376054, -1.298763, -2.625084, -0.788543, 1.570796, 1.946850],accel_mss,speed_ms,0,blend_radius_m)
    movel([0.376104, -1.298048, -2.625508, -0.788833, 1.570796, 1.946900],accel_mss,speed_ms,0,blend_radius_m)
    movel([0.376079, -1.297325, -2.625936, -0.789128, 1.570796, 1.946875],accel_mss,speed_ms,0,blend_radius_m)
    speed_ms = 0.005
    movel([0.376079, -1.288096, -2.621565, -0.802728, 1.570796, 1.946875],accel_mss,speed_ms,0,blend_radius_m)
    speed_ms = 0.040
    movel([0.373085, -1.283236, -2.624389, -0.804764, 1.570796, 1.943881],accel_mss,speed_ms,0,blend_radius_m)
    speed_ms = 0.005
    movel([0.373085, -1.292491, -2.628783, -0.791115, 1.570796, 1.943881],accel_mss,speed_ms,0,blend_radius_m)
    speed_ms = 0.025
    movel([0.373833, -1.292874, -2.628559, -0.790957, 1.570796, 1.944630],accel_mss,speed_ms,0,blend_radius_m)
    movel([0.372980, -1.292866, -2.628563, -0.790960, 1.570796, 1.943776],accel_mss,speed_ms,0,blend_radius_m)
    movel([0.371335, -1.292845, -2.628576, -0.790969, 1.570796, 1.942131],accel_mss,speed_ms,0,blend_radius_m)
    movel([0.369247, -1.293140, -2.628402, -0.790847, 1.570796, 1.940044],accel_mss,speed_ms,0,blend_radius_m)
    movel([0.366745, -1.293745, -2.628047, -0.790597, 1.570796, 1.937542],accel_mss,speed_ms,0,blend_radius_m)
    movel([0.361830, -1.295297, -2.627134, -0.789958, 1.570796, 1.932626],accel_mss,speed_ms,0,blend_radius_m)
    movel([0.360475, -1.295574, -2.626971, -0.789844, 1.570796, 1.931272],accel_mss,speed_ms,0,blend_radius_m)
    movel([0.359516, -1.295549, -2.626986, -0.789855, 1.570796, 1.930313],accel_mss,speed_ms,0,blend_radius_m)
    movel([0.358798, -1.295235, -2.627171, -0.789983, 1.570796, 1.929595],accel_mss,speed_ms,0,blend_radius_m)
    movel([0.358332, -1.294773, -2.627443, -0.790173, 1.570796, 1.929129],accel_mss,speed_ms,0,blend_radius_m)
    movel([0.358133, -1.294512, -2.627596, -0.790281, 1.570796, 1.928929],accel_mss,speed_ms,0,blend_radius_m)
    movel([0.357867, -1.293874, -2.627971, -0.790544, 1.570796, 1.928664],accel_mss,speed_ms,0,blend_radius_m)
    movel([0.359697, -1.294459, -2.627628, -0.790302, 1.570796, 1.930493],accel_mss,speed_ms,0,blend_radius_m)
    movel([0.360240, -1.294520, -2.627592, -0.790278, 1.570796, 1.931037],accel_mss,speed_ms,0,blend_radius_m)
    movel([0.363439, -1.294273, -2.627737, -0.790379, 1.570796, 1.934235],accel_mss,speed_ms,0,blend_radius_m)
    movel([0.364308, -1.294112, -2.627831, -0.790445, 1.570796, 1.935105],accel_mss,speed_ms,0,blend_radius_m)
    movel([0.366683, -1.293315, -2.628299, -0.790774, 1.570796, 1.937479],accel_mss,speed_ms,0,blend_radius_m)
    movel([0.368798, -1.292618, -2.628709, -0.791063, 1.570796, 1.939594],accel_mss,speed_ms,0,blend_radius_m)
    movel([0.370540, -1.292253, -2.628922, -0.791214, 1.570796, 1.941336],accel_mss,speed_ms,0,blend_radius_m)
    movel([0.371956, -1.292215, -2.628945, -0.791230, 1.570796, 1.942753],accel_mss,speed_ms,0,blend_radius_m)
    movel([0.373085, -1.292491, -2.628783, -0.791115, 1.570796, 1.943881],accel_mss,speed_ms,0,blend_radius_m)
    movel([0.373833, -1.292874, -2.628559, -0.790957, 1.570796, 1.944630],accel_mss,speed_ms,0,blend_radius_m)
    movel([0.372980, -1.292866, -2.628563, -0.790960, 1.570796, 1.943776],accel_mss,speed_ms,0,blend_radius_m)
    movel([0.372322, -1.292858, -2.628568, -0.790963, 1.570796, 1.943119],accel_mss,speed_ms,0,blend_radius_m)
    speed_ms = 0.005
    movel([0.372322, -1.283604, -2.624176, -0.804609, 1.570796, 1.943119],accel_mss,speed_ms,0,blend_radius_m)
    speed_ms = 0.040
    movel([0.360909, -1.274556, -2.629359, -0.808474, 1.570796, 1.931705],accel_mss,speed_ms,0,blend_radius_m)
    speed_ms = 0.005
    movel([0.360909, -1.283859, -2.633792, -0.794738, 1.570796, 1.931705],accel_mss,speed_ms,0,blend_radius_m)
    speed_ms = 0.025
    movel([0.361097, -1.281306, -2.635255, -0.795828, 1.570796, 1.931893],accel_mss,speed_ms,0,blend_radius_m)
    movel([0.361051, -1.280052, -2.635971, -0.796366, 1.570796, 1.931847],accel_mss,speed_ms,0,blend_radius_m)
    movel([0.360898, -1.279299, -2.636399, -0.796690, 1.570796, 1.931695],accel_mss,speed_ms,0,blend_radius_m)
    movel([0.360676, -1.278855, -2.636652, -0.796882, 1.570796, 1.931472],accel_mss,speed_ms,0,blend_radius_m)
    movel([0.360391, -1.278613, -2.636790, -0.796986, 1.570796, 1.931187],accel_mss,speed_ms,0,blend_radius_m)
    movel([0.360087, -1.278597, -2.636799, -0.796993, 1.570796, 1.930883],accel_mss,speed_ms,0,blend_radius_m)
    movel([0.359475, -1.279029, -2.636553, -0.796806, 1.570796, 1.930271],accel_mss,speed_ms,0,blend_radius_m)
    movel([0.359149, -1.279096, -2.636515, -0.796778, 1.570796, 1.929945],accel_mss,speed_ms,0,blend_radius_m)
    movel([0.358083, -1.278514, -2.636846, -0.797029, 1.570796, 1.928880],accel_mss,speed_ms,0,blend_radius_m)
    movel([0.357471, -1.278107, -2.637077, -0.797205, 1.570796, 1.928268],accel_mss,speed_ms,0,blend_radius_m)
    movel([0.357048, -1.277945, -2.637169, -0.797275, 1.570796, 1.927844],accel_mss,speed_ms,0,blend_radius_m)
    movel([0.356669, -1.277958, -2.637162, -0.797269, 1.570796, 1.927465],accel_mss,speed_ms,0,blend_radius_m)
    movel([0.356256, -1.278133, -2.637062, -0.797194, 1.570796, 1.927052],accel_mss,speed_ms,0,blend_radius_m)
    movel([0.356037, -1.278442, -2.636887, -0.797060, 1.570796, 1.926833],accel_mss,speed_ms,0,blend_radius_m)
    movel([0.356089, -1.278977, -2.636583, -0.796829, 1.570796, 1.926886],accel_mss,speed_ms,0,blend_radius_m)
    movel([0.356368, -1.279627, -2.636213, -0.796549, 1.570796, 1.927164],accel_mss,speed_ms,0,blend_radius_m)
    movel([0.357293, -1.280992, -2.635434, -0.795962, 1.570796, 1.928090],accel_mss,speed_ms,0,blend_radius_m)
    movel([0.357278, -1.281289, -2.635265, -0.795835, 1.570796, 1.928074],accel_mss,speed_ms,0,blend_radius_m)
    movel([0.356815, -1.282452, -2.634599, -0.795338, 1.570796, 1.927612],accel_mss,speed_ms,0,blend_radius_m)
    movel([0.357850, -1.282624, -2.634501, -0.795264, 1.570796, 1.928647],accel_mss,speed_ms,0,blend_radius_m)
    movel([0.358872, -1.282706, -2.634454, -0.795229, 1.570796, 1.929669],accel_mss,speed_ms,0,blend_radius_m)
    movel([0.358939, -1.280975, -2.635444, -0.795970, 1.570796, 1.929735],accel_mss,speed_ms,0,blend_radius_m)
    movel([0.358982, -1.280701, -2.635601, -0.796087, 1.570796, 1.929779],accel_mss,speed_ms,0,blend_radius_m)
    movel([0.359359, -1.280259, -2.635853, -0.796277, 1.570796, 1.930155],accel_mss,speed_ms,0,blend_radius_m)
    movel([0.359630, -1.280060, -2.635967, -0.796363, 1.570796, 1.930427],accel_mss,speed_ms,0,blend_radius_m)
    movel([0.359871, -1.280071, -2.635960, -0.796358, 1.570796, 1.930667],accel_mss,speed_ms,0,blend_radius_m)
    movel([0.360000, -1.280308, -2.635825, -0.796256, 1.570796, 1.930796],accel_mss,speed_ms,0,blend_radius_m)
    movel([0.360158, -1.281026, -2.635415, -0.795948, 1.570796, 1.930954],accel_mss,speed_ms,0,blend_radius_m)
    movel([0.360117, -1.282337, -2.634665, -0.795387, 1.570796, 1.930913],accel_mss,speed_ms,0,blend_radius_m)
    movel([0.359973, -1.283681, -2.633894, -0.794814, 1.570796, 1.930769],accel_mss,speed_ms,0,blend_radius_m)
    movel([0.359706, -1.284183, -2.633605, -0.794600, 1.570796, 1.930502],accel_mss,speed_ms,0,blend_radius_m)
    movel([0.359553, -1.284531, -2.633405, -0.794453, 1.570796, 1.930349],accel_mss,speed_ms,0,blend_radius_m)
    movel([0.359665, -1.284681, -2.633319, -0.794389, 1.570796, 1.930461],accel_mss,speed_ms,0,blend_radius_m)
    movel([0.360589, -1.285200, -2.633020, -0.794169, 1.570796, 1.931386],accel_mss,speed_ms,0,blend_radius_m)
    movel([0.360909, -1.283859, -2.633792, -0.794738, 1.570796, 1.931705],accel_mss,speed_ms,0,blend_radius_m)
    movel([0.361092, -1.281386, -2.635209, -0.795794, 1.570796, 1.931889],accel_mss,speed_ms,0,blend_radius_m)
    speed_ms = 0.005
    movel([0.361092, -1.272070, -2.630766, -0.809554, 1.570796, 1.931889],accel_mss,speed_ms,0,blend_radius_m)
    speed_ms = 0.040
    movel([0.352046, -1.270244, -2.631793, -0.810352, 1.570796, 1.922843],accel_mss,speed_ms,0,blend_radius_m)
    speed_ms = 0.005
    movel([0.352046, -1.279570, -2.636246, -0.796574, 1.570796, 1.922843],accel_mss,speed_ms,0,blend_radius_m)
    speed_ms = 0.025
    movel([0.350726, -1.280552, -2.635686, -0.796151, 1.570796, 1.921522],accel_mss,speed_ms,0,blend_radius_m)
    movel([0.350409, -1.280755, -2.635570, -0.796064, 1.570796, 1.921205],accel_mss,speed_ms,0,blend_radius_m)
    movel([0.349573, -1.281438, -2.635180, -0.795771, 1.570796, 1.920369],accel_mss,speed_ms,0,blend_radius_m)
    movel([0.349367, -1.281688, -2.635037, -0.795664, 1.570796, 1.920163],accel_mss,speed_ms,0,blend_radius_m)
    movel([0.349281, -1.282014, -2.634850, -0.795525, 1.570796, 1.920078],accel_mss,speed_ms,0,blend_radius_m)
    movel([0.349376, -1.282211, -2.634737, -0.795441, 1.570796, 1.920172],accel_mss,speed_ms,0,blend_radius_m)
    movel([0.349450, -1.282722, -2.634445, -0.795223, 1.570796, 1.920246],accel_mss,speed_ms,0,blend_radius_m)
    movel([0.349219, -1.283722, -2.633871, -0.794797, 1.570796, 1.920015],accel_mss,speed_ms,0,blend_radius_m)
    movel([0.348833, -1.284811, -2.633244, -0.794334, 1.570796, 1.919629],accel_mss,speed_ms,0,blend_radius_m)
    movel([0.348360, -1.285691, -2.632736, -0.793961, 1.570796, 1.919156],accel_mss,speed_ms,0,blend_radius_m)
    movel([0.346176, -1.288603, -2.631050, -0.792735, 1.570796, 1.916973],accel_mss,speed_ms,0,blend_radius_m)
    movel([0.345853, -1.288937, -2.630857, -0.792595, 1.570796, 1.916649],accel_mss,speed_ms,0,blend_radius_m)
    movel([0.345592, -1.289084, -2.630771, -0.792534, 1.570796, 1.916388],accel_mss,speed_ms,0,blend_radius_m)
    movel([0.345282, -1.289128, -2.630746, -0.792515, 1.570796, 1.916078],accel_mss,speed_ms,0,blend_radius_m)
    movel([0.344779, -1.289269, -2.630664, -0.792457, 1.570796, 1.915576],accel_mss,speed_ms,0,blend_radius_m)
    movel([0.344577, -1.289528, -2.630513, -0.792348, 1.570796, 1.915373],accel_mss,speed_ms,0,blend_radius_m)
    movel([0.343400, -1.291475, -2.629377, -0.791537, 1.570796, 1.914196],accel_mss,speed_ms,0,blend_radius_m)
    movel([0.342359, -1.292811, -2.628595, -0.790983, 1.570796, 1.913155],accel_mss,speed_ms,0,blend_radius_m)
    movel([0.341234, -1.294031, -2.627879, -0.790479, 1.570796, 1.912031],accel_mss,speed_ms,0,blend_radius_m)
    movel([0.340185, -1.294941, -2.627344, -0.790104, 1.570796, 1.910981],accel_mss,speed_ms,0,blend_radius_m)
    movel([0.339211, -1.295614, -2.626947, -0.789828, 1.570796, 1.910007],accel_mss,speed_ms,0,blend_radius_m)
    movel([0.338682, -1.295791, -2.626843, -0.789755, 1.570796, 1.909478],accel_mss,speed_ms,0,blend_radius_m)
    movel([0.338447, -1.295587, -2.626963, -0.789839, 1.570796, 1.909243],accel_mss,speed_ms,0,blend_radius_m)
    movel([0.338512, -1.294948, -2.627340, -0.790101, 1.570796, 1.909309],accel_mss,speed_ms,0,blend_radius_m)
    movel([0.338713, -1.294120, -2.627827, -0.790442, 1.570796, 1.909510],accel_mss,speed_ms,0,blend_radius_m)
    movel([0.338129, -1.294814, -2.627419, -0.790156, 1.570796, 1.908925],accel_mss,speed_ms,0,blend_radius_m)
    movel([0.335286, -1.297812, -2.625648, -0.788929, 1.570796, 1.906082],accel_mss,speed_ms,0,blend_radius_m)
    movel([0.333596, -1.299421, -2.624693, -0.788275, 1.570796, 1.904392],accel_mss,speed_ms,0,blend_radius_m)
    movel([0.330932, -1.301652, -2.623363, -0.787375, 1.570796, 1.901728],accel_mss,speed_ms,0,blend_radius_m)
    movel([0.330138, -1.302174, -2.623051, -0.787165, 1.570796, 1.900934],accel_mss,speed_ms,0,blend_radius_m)
    movel([0.329651, -1.302339, -2.622952, -0.787098, 1.570796, 1.900448],accel_mss,speed_ms,0,blend_radius_m)
    movel([0.329404, -1.302208, -2.623030, -0.787151, 1.570796, 1.900200],accel_mss,speed_ms,0,blend_radius_m)
    movel([0.329712, -1.301575, -2.623409, -0.787406, 1.570796, 1.900508],accel_mss,speed_ms,0,blend_radius_m)
    movel([0.330081, -1.300968, -2.623771, -0.787650, 1.570796, 1.900877],accel_mss,speed_ms,0,blend_radius_m)
    movel([0.331306, -1.299082, -2.624894, -0.788413, 1.570796, 1.902102],accel_mss,speed_ms,0,blend_radius_m)
    movel([0.331670, -1.298377, -2.625312, -0.788699, 1.570796, 1.902467],accel_mss,speed_ms,0,blend_radius_m)
    movel([0.332580, -1.295268, -2.627151, -0.789970, 1.570796, 1.903377],accel_mss,speed_ms,0,blend_radius_m)
    movel([0.332687, -1.295094, -2.627254, -0.790041, 1.570796, 1.903483],accel_mss,speed_ms,0,blend_radius_m)
    movel([0.333051, -1.294898, -2.627369, -0.790122, 1.570796, 1.903847],accel_mss,speed_ms,0,blend_radius_m)
    movel([0.333400, -1.294997, -2.627311, -0.790081, 1.570796, 1.904196],accel_mss,speed_ms,0,blend_radius_m)
    movel([0.333513, -1.295473, -2.627031, -0.789886, 1.570796, 1.904310],accel_mss,speed_ms,0,blend_radius_m)
    movel([0.333369, -1.296352, -2.626512, -0.789526, 1.570796, 1.904165],accel_mss,speed_ms,0,blend_radius_m)
    movel([0.332468, -1.299246, -2.624796, -0.788346, 1.570796, 1.903264],accel_mss,speed_ms,0,blend_radius_m)
    movel([0.333060, -1.298841, -2.625038, -0.788511, 1.570796, 1.903857],accel_mss,speed_ms,0,blend_radius_m)
    movel([0.334701, -1.297178, -2.626023, -0.789188, 1.570796, 1.905498],accel_mss,speed_ms,0,blend_radius_m)
    movel([0.339129, -1.292381, -2.628847, -0.791161, 1.570796, 1.909925],accel_mss,speed_ms,0,blend_radius_m)
    movel([0.339470, -1.292099, -2.629012, -0.791278, 1.570796, 1.910266],accel_mss,speed_ms,0,blend_radius_m)
    movel([0.339852, -1.291915, -2.629120, -0.791354, 1.570796, 1.910648],accel_mss,speed_ms,0,blend_radius_m)
    movel([0.340105, -1.291922, -2.629116, -0.791351, 1.570796, 1.910901],accel_mss,speed_ms,0,blend_radius_m)
    movel([0.340213, -1.292101, -2.629011, -0.791277, 1.570796, 1.911009],accel_mss,speed_ms,0,blend_radius_m)
    movel([0.340131, -1.293204, -2.628365, -0.790820, 1.570796, 1.910927],accel_mss,speed_ms,0,blend_radius_m)
    movel([0.340095, -1.293842, -2.627990, -0.790557, 1.570796, 1.910891],accel_mss,speed_ms,0,blend_radius_m)
    movel([0.340385, -1.293737, -2.628052, -0.790600, 1.570796, 1.911181],accel_mss,speed_ms,0,blend_radius_m)
    movel([0.341029, -1.293046, -2.628457, -0.790885, 1.570796, 1.911825],accel_mss,speed_ms,0,blend_radius_m)
    movel([0.342320, -1.291451, -2.629392, -0.791547, 1.570796, 1.913117],accel_mss,speed_ms,0,blend_radius_m)
    movel([0.342678, -1.290913, -2.629706, -0.791771, 1.570796, 1.913474],accel_mss,speed_ms,0,blend_radius_m)
    movel([0.344707, -1.287200, -2.631864, -0.793325, 1.570796, 1.915504],accel_mss,speed_ms,0,blend_radius_m)
    movel([0.345022, -1.286686, -2.632162, -0.793541, 1.570796, 1.915819],accel_mss,speed_ms,0,blend_radius_m)
    movel([0.345276, -1.286420, -2.632316, -0.793654, 1.570796, 1.916072],accel_mss,speed_ms,0,blend_radius_m)
    movel([0.345565, -1.286274, -2.632400, -0.793715, 1.570796, 1.916361],accel_mss,speed_ms,0,blend_radius_m)
    movel([0.345919, -1.286308, -2.632380, -0.793701, 1.570796, 1.916715],accel_mss,speed_ms,0,blend_radius_m)
    movel([0.345989, -1.286458, -2.632294, -0.793638, 1.570796, 1.916786],accel_mss,speed_ms,0,blend_radius_m)
    movel([0.346060, -1.287092, -2.631927, -0.793370, 1.570796, 1.916857],accel_mss,speed_ms,0,blend_radius_m)
    movel([0.346199, -1.287137, -2.631901, -0.793351, 1.570796, 1.916995],accel_mss,speed_ms,0,blend_radius_m)
    movel([0.346613, -1.286673, -2.632169, -0.793547, 1.570796, 1.917409],accel_mss,speed_ms,0,blend_radius_m)
    movel([0.347721, -1.284766, -2.633270, -0.794353, 1.570796, 1.918517],accel_mss,speed_ms,0,blend_radius_m)
    movel([0.348015, -1.284034, -2.633691, -0.794664, 1.570796, 1.918811],accel_mss,speed_ms,0,blend_radius_m)
    movel([0.348173, -1.283275, -2.634127, -0.794987, 1.570796, 1.918969],accel_mss,speed_ms,0,blend_radius_m)
    movel([0.348061, -1.283203, -2.634169, -0.795018, 1.570796, 1.918858],accel_mss,speed_ms,0,blend_radius_m)
    movel([0.347358, -1.283201, -2.634170, -0.795018, 1.570796, 1.918154],accel_mss,speed_ms,0,blend_radius_m)
    movel([0.347299, -1.282914, -2.634334, -0.795141, 1.570796, 1.918095],accel_mss,speed_ms,0,blend_radius_m)
    movel([0.347686, -1.282282, -2.634697, -0.795411, 1.570796, 1.918482],accel_mss,speed_ms,0,blend_radius_m)
    movel([0.348658, -1.281144, -2.635348, -0.795897, 1.570796, 1.919454],accel_mss,speed_ms,0,blend_radius_m)
    movel([0.350016, -1.279729, -2.636155, -0.796505, 1.570796, 1.920812],accel_mss,speed_ms,0,blend_radius_m)
    movel([0.350378, -1.279523, -2.636273, -0.796594, 1.570796, 1.921174],accel_mss,speed_ms,0,blend_radius_m)
